								FOR j:= Iforstart TO Iforend DO
									IF NOT HMI_WorkAreaDataPicking[j].Destinazione THEN
										IF HMI_WorkAreaDataPicking[j].NumElementiDaLavorare >= 1 THEN
											ElementiDaDepositare[IdxLista] := ElementiElaborati[IdxLista] + HMI_WorkAreaDataPicking[j].NumElementiDaLavorare;
											FOR k := ElementiElaborati[IdxLista] TO ElementiDaDepositare[IdxLista]-1 DO	
												WorkAreaProductionList[NumPostazioneDeposito].PElementList[k].WA_PRELIEVO := j;
												WorkAreaProductionList[NumPostazioneDeposito].PElementList[k].WA_DEPOSITO := i;	
												ElementiElaborati[IdxLista] := ElementiElaborati[IdxLista]+1; 
											END_FOR
											CASE HMI_WorkAreaDataPicking[j].Typology OF 
												(* Se ho una cassa pianale in legno *)
												LEGNO_PIANO:
													WorkAreaState[j].Supporto.Code 					:= ActualPickingListFromHMI[IdxLista].SupportPianoLegno.Code;
													WorkAreaState[j].Supporto.DimBaseUtile		 	:= ActualPickingListFromHMI[IdxLista].SupportPianoLegno.DimBaseUtile;
													WorkAreaState[j].Supporto.AltezzaDenteRitenuta 	:= ActualPickingListFromHMI[IdxLista].SupportPianoLegno.ZDim+20;
													WorkAreaState[j].Supporto.DimVertice 			:= ActualPickingListFromHMI[IdxLista].SupportPianoLegno.DimVertice;
													WorkAreaState[j].Supporto.HMAX 					:= ActualPickingListFromHMI[IdxLista].SupportPianoLegno.HMAX;
													WorkAreaState[j].Supporto.Tipologia 			:=  e_Tipo_Pallet.CASSA_STANDARD;//ActualPickingListFromHMI[1].Support.Tipologia;
													WorkAreaState[j].Supporto.XDim 					:= ActualPickingListFromHMI[IdxLista].SupportPianoLegno.XDim;
													WorkAreaState[j].Supporto.YDim 					:= ActualPickingListFromHMI[IdxLista].SupportPianoLegno.YDim;
													WorkAreaState[j].Supporto.ZDim 					:= ActualPickingListFromHMI[IdxLista].SupportPianoLegno.ZDim;
													WorkAreaOffset[j].Y 							:= OFFSET_POSTAZIONE_LEGNO + ActualPickingListFromHMI[IdxLista].SupportPianoLegno.YDim/2;//ATTENZIONE!!! per poter lavorare in centro con i supporti pari, questa misura è la distanza tra il riscontro bundle verticale e il centro postazione PARI
												(* Se ho una cassa pianale in ferro su supporto *)
												TELAIO_PIANO:
													WorkAreaState[j].Supporto.Code 					:= ActualPickingListFromHMI[IdxLista].SupportPianoFerro.Code;
													WorkAreaState[j].Supporto.DimBaseUtile		 	:= ActualPickingListFromHMI[IdxLista].SupportPianoFerro.DimBaseUtile;
													WorkAreaState[j].Supporto.AltezzaDenteRitenuta 	:= ActualPickingListFromHMI[IdxLista].SupportPianoFerro.ZDim+20;
													WorkAreaState[j].Supporto.DimVertice 			:= ActualPickingListFromHMI[IdxLista].SupportPianoFerro.DimVertice;
													WorkAreaState[j].Supporto.HMAX 					:= ActualPickingListFromHMI[IdxLista].SupportPianoFerro.HMAX;
													WorkAreaState[j].Supporto.Tipologia 			:=  e_Tipo_Pallet.CASSA_STANDARD;//ActualPickingListFromHMI[1].Support.Tipologia;
													WorkAreaState[j].Supporto.XDim 					:= ActualPickingListFromHMI[IdxLista].SupportPianoFerro.XDim;
													WorkAreaState[j].Supporto.YDim 					:= ActualPickingListFromHMI[IdxLista].SupportPianoFerro.YDim;
													WorkAreaState[j].Supporto.ZDim 					:= ActualPickingListFromHMI[IdxLista].SupportPianoFerro.ZDim;
													WorkAreaOffset[j].Y 							:= OFFSET_POSTAZIONE_TELAIO - ActualPickingListFromHMI[IdxLista].SupportPianoFerro.YDim/2;//ATTENZIONE!!! per poter lavorare in centro con i supporti pari, questa misura è la distanza tra il riscontro bundle verticale e il centro postazione PARI
												(* Se ho un bundle *)
												BUNDLE_VERT:
													//WorkAreaState[j].P := ElementiDaDepositare;
													WorkAreaState[j].Supporto.Code 					:= ActualPickingListFromHMI[IdxLista].SupportVertBundle.Code;
													WorkAreaState[j].Supporto.DimBaseUtile		 	:= ActualPickingListFromHMI[IdxLista].SupportVertBundle.DimBaseUtile;
													WorkAreaState[j].Supporto.AltezzaDenteRitenuta 	:= ActualPickingListFromHMI[IdxLista].SupportVertBundle.ZDim+20;
													WorkAreaState[j].Supporto.DimVertice 			:= ActualPickingListFromHMI[IdxLista].SupportVertBundle.DimVertice;
													WorkAreaState[j].Supporto.HMAX 					:= ActualPickingListFromHMI[IdxLista].SupportVertBundle.HMAX;
													WorkAreaState[j].Supporto.Tipologia 			:= e_Tipo_Pallet.BUNDLE;//ActualPickingListFromHMI.SupportVertBundle.Tipologia;
													WorkAreaState[j].Supporto.XDim 					:= ActualPickingListFromHMI[IdxLista].SupportVertBundle.XDim;
													WorkAreaState[j].Supporto.YDim 					:= ActualPickingListFromHMI[IdxLista].SupportVertBundle.YDim;
													WorkAreaState[j].Supporto.ZDim 					:= ActualPickingListFromHMI[IdxLista].SupportVertBundle.ZDim;
													WorkAreaState[j].Supporto.ZDim_Ext1        		:= WorkAreaState[j].Supporto.ZDim + 20;	
													 WorkAreaOffset[j].Y 		:= 0 ;	
													//Mod 25/&/2025	  
													//WorkAreaOffset[j].Y 		:= ActualPickingListFromHMI[IdxLista].SupportVertBundle.YDim-ActualPickingListFromHMI[IdxLista].SupportVertBundle.DimBaseUtile -40;				
												(* Se ho un A_Frame *)	  
												A_FRAME_VERT:  						
													//WorkAreaState[j].P := ElementiDaDepositare;
													WorkAreaState[j].Supporto.Code 					:= ActualPickingListFromHMI[IdxLista].SupportVertCav.Code;
													WorkAreaState[j].Supporto.DimBaseUtile		 	:= ActualPickingListFromHMI[IdxLista].SupportVertCav.DimBaseUtile;
													WorkAreaState[j].Supporto.AltezzaDenteRitenuta 	:= ActualPickingListFromHMI[IdxLista].SupportVertCav.ZDim+20;
													WorkAreaState[j].Supporto.DimVertice 			:= ActualPickingListFromHMI[IdxLista].SupportVertCav.DimVertice;
													WorkAreaState[j].Supporto.HMAX 					:= ActualPickingListFromHMI[IdxLista].SupportVertcav.HMAX;
													WorkAreaState[j].Supporto.Tipologia 			:= CAVALLETTO;//ActualPickingListFromHMI.SupportVert.Tipologia;
													WorkAreaState[j].Supporto.XDim 					:= ActualPickingListFromHMI[IdxLista].SupportVertCav.XDim;
													WorkAreaState[j].Supporto.YDim 					:= ActualPickingListFromHMI[IdxLista].SupportVertCav.YDim;
													WorkAreaState[j].Supporto.ZDim 					:= ActualPickingListFromHMI[IdxLista].SupportVertCav.ZDim;
													WorkAreaState[j].Supporto.ZDim_Ext1        		:= WorkAreaState[j].Supporto.ZDim + 20;		
													WorkAreaOffset[j].Y 							:= OFFSET_POSTAZIONE_LEGNO + ActualPickingListFromHMI[IdxLista].SupportVertCav.YDim/2;//ATTENZIONE!!! per poter lavorare in centro con i supporti pari, questa misura è la distanza tra il riscontro bundle verticale e il centro postazione PARI
											   		CoordenadaPasillo0_Y := WorkArea[j].Y +  WorkAreaOffset[j].Y  - Dimensioni_Pinza.Spessore - INGOMBRO_RISCONTRO_BUNDLE - WorkAreaState[j].Supporto.YDim /2 ;
													CoordenadaPasillo180_Y := WorkArea[j].Y + WorkAreaState[j].Supporto.YDim /2 + WorkAreaOffset[j].Y  + Dimensioni_Pinza.Spessore + INGOMBRO_RISCONTRO_FRAME  ;	
											END_CASE	
											WorkAreaProductionList[j].Support := HMI_Formatura.HMI_Forming_Supporto; 
										END_IF
									END_IF     
									TFClearApprendimento(ADR(WorkAreaState[j].Apprendimento));//Azzeramento apprendimento 
								END_FOR
								EXIT; 
							(* Se ho un bundle *)
							BUNDLE_VERT:
								CASE HMI_WorkAreaDataPicking[NumPostazioneDeposito].Typology OF
									LEGNO_PIANO:
										 		WorkAreaProductionList[NumPostazioneDeposito].Support := WorkAreaState[NumPostazioneDeposito].Supporto;
												WorkAreaProductionList[NumPostazioneDeposito].Support.Tipologia	:= e_Tipo_Pallet.CASSA_STANDARD; 
									TELAIO_PIANO:
										 		WorkAreaProductionList[NumPostazioneDeposito].Support := WorkAreaState[NumPostazioneDeposito].Supporto;
												WorkAreaProductionList[NumPostazioneDeposito].Support.Tipologia	:= e_Tipo_Pallet.CASSA_STANDARD; 
									BUNDLE_VERT:
										 		WorkAreaProductionList[NumPostazioneDeposito].Support := WorkAreaState[NumPostazioneDeposito].Supporto;
												WorkAreaProductionList[NumPostazioneDeposito].Support.Tipologia	:= e_Tipo_Pallet.BUNDLE; 
									A_FRAME_VERT:
										 		WorkAreaProductionList[NumPostazioneDeposito].Support := WorkAreaState[NumPostazioneDeposito].Supporto;
												WorkAreaProductionList[NumPostazioneDeposito].Support.Tipologia	:= e_Tipo_Pallet.CAVALLETTO; 
								END_CASE
								//Se ho deposito verticale su bundle
								WorkAreaState[NumPostazioneDeposito].Supporto.Code 						:= ActualPickingListFromHMI[IdxLista].SupportVertBundle.Code;
								WorkAreaState[NumPostazioneDeposito].Supporto.DimBaseUtile		 		:= ActualPickingListFromHMI[IdxLista].SupportVertBundle.DimBaseUtile;
								WorkAreaState[NumPostazioneDeposito].Supporto.DimVertice 				:= ActualPickingListFromHMI[IdxLista].SupportVertBundle.DimVertice;
								WorkAreaState[NumPostazioneDeposito].Supporto.HMAX 						:= ActualPickingListFromHMI[IdxLista].SupportVertBundle.HMAX;
								WorkAreaState[NumPostazioneDeposito].Supporto.Tipologia 				:= e_Tipo_Pallet.BUNDLE;
								WorkAreaState[NumPostazioneDeposito].Supporto.XDim 						:= ActualPickingListFromHMI[IdxLista].SupportVertBundle.XDim;
								WorkAreaState[NumPostazioneDeposito].Supporto.YDim 						:= ActualPickingListFromHMI[IdxLista].SupportVertBundle.YDim;
								WorkAreaState[NumPostazioneDeposito].Supporto.ZDim 						:= ActualPickingListFromHMI[IdxLista].SupportVertBundle.ZDim;
								//Lo que HABIA
								//PruevaWorkAreaOffset[NumPostazioneDeposito].Y 								:= -40;	
								//Mod 25/&/2025	  
								//WorkAreaOffset[NumPostazioneDeposito].Y 								:= ActualPickingListFromHMI[IdxLista].SupportVertBundle.YDim-ActualPickingListFromHMI[IdxLista].SupportVertBundle.DimBaseUtile -20;
								FOR j:= Iforstart TO Iforend DO
									IF NOT HMI_WorkAreaDataPicking[j].Destinazione THEN
										IF HMI_WorkAreaDataPicking[j].NumElementiDaLavorare >= 1 THEN
											ElementiDaDepositare[IdxLista] := ElementiElaborati[IdxLista] + HMI_WorkAreaDataPicking[j].NumElementiDaLavorare;
											FOR k := ElementiElaborati[IdxLista] TO ElementiDaDepositare[IdxLista]-1 DO	
												WorkAreaProductionList[NumPostazioneDeposito].PElementList[k].WA_PRELIEVO := j;
												WorkAreaProductionList[NumPostazioneDeposito].PElementList[k].WA_DEPOSITO := i;	
												ElementiElaborati[IdxLista] := ElementiElaborati[IdxLista]+1; 
											END_FOR
											CASE HMI_WorkAreaDataPicking[j].Typology OF 
												(* Se ho una cassa pianale in legno *)
												LEGNO_PIANO:
													WorkAreaState[j].Supporto.Code 					:= ActualPickingListFromHMI[IdxLista].SupportPianoLegno.Code;
													WorkAreaState[j].Supporto.DimBaseUtile		 	:= ActualPickingListFromHMI[IdxLista].SupportPianoLegno.DimBaseUtile;
													WorkAreaState[j].Supporto.AltezzaDenteRitenuta 	:= ActualPickingListFromHMI[IdxLista].SupportPianoLegno.ZDim+20;
													WorkAreaState[j].Supporto.DimVertice 			:= ActualPickingListFromHMI[IdxLista].SupportPianoLegno.DimVertice;
													WorkAreaState[j].Supporto.HMAX 					:= ActualPickingListFromHMI[IdxLista].SupportPianoLegno.HMAX;
													WorkAreaState[j].Supporto.Tipologia 			:=  e_Tipo_Pallet.CASSA_STANDARD;//ActualPickingListFromHMI[1].Support.Tipologia;
													WorkAreaState[j].Supporto.XDim 					:= ActualPickingListFromHMI[IdxLista].SupportPianoLegno.XDim;
													WorkAreaState[j].Supporto.YDim 					:= ActualPickingListFromHMI[IdxLista].SupportPianoLegno.YDim;
													WorkAreaState[j].Supporto.ZDim 					:= ActualPickingListFromHMI[IdxLista].SupportPianoLegno.ZDim;
													WorkAreaOffset[j].Y 							:= OFFSET_POSTAZIONE_LEGNO + ActualPickingListFromHMI[IdxLista].SupportPianoLegno.YDim/2;//ATTENZIONE!!! per poter lavorare in centro con i supporti pari, questa misura è la distanza tra il riscontro bundle verticale e il centro postazione PARI
												(* Se ho una cassa pianale in ferro su supporto *)
												TELAIO_PIANO:
													WorkAreaState[j].Supporto.Code 					:= ActualPickingListFromHMI[IdxLista].SupportPianoFerro.Code;
													WorkAreaState[j].Supporto.DimBaseUtile		 	:= ActualPickingListFromHMI[IdxLista].SupportPianoFerro.DimBaseUtile;
													WorkAreaState[j].Supporto.AltezzaDenteRitenuta 	:= ActualPickingListFromHMI[IdxLista].SupportPianoFerro.ZDim+20;
													WorkAreaState[j].Supporto.DimVertice 			:= ActualPickingListFromHMI[IdxLista].SupportPianoFerro.DimVertice;
													WorkAreaState[j].Supporto.HMAX 					:= ActualPickingListFromHMI[IdxLista].SupportPianoFerro.HMAX;
													WorkAreaState[j].Supporto.Tipologia 			:=  e_Tipo_Pallet.CASSA_STANDARD;//ActualPickingListFromHMI[1].Support.Tipologia;
													WorkAreaState[j].Supporto.XDim 					:= ActualPickingListFromHMI[IdxLista].SupportPianoFerro.XDim;
													WorkAreaState[j].Supporto.YDim 					:= ActualPickingListFromHMI[IdxLista].SupportPianoFerro.YDim;
													WorkAreaState[j].Supporto.ZDim 					:= ActualPickingListFromHMI[IdxLista].SupportPianoFerro.ZDim;
													WorkAreaOffset[j].Y 							:= OFFSET_POSTAZIONE_TELAIO - ActualPickingListFromHMI[IdxLista].SupportPianoFerro.YDim/2;//ATTENZIONE!!! per poter lavorare in centro con i supporti pari, questa misura è la distanza tra il riscontro bundle verticale e il centro postazione PARI
												(* Se ho un bundle *)
												BUNDLE_VERT:
													//WorkAreaState[j].P := ElementiDaDepositare;
													WorkAreaState[j].Supporto.Code 					:= ActualPickingListFromHMI[IdxLista].SupportVertBundle.Code;
													WorkAreaState[j].Supporto.DimBaseUtile		 	:= ActualPickingListFromHMI[IdxLista].SupportVertBundle.DimBaseUtile;
													WorkAreaState[j].Supporto.AltezzaDenteRitenuta 	:= ActualPickingListFromHMI[IdxLista].SupportVertBundle.ZDim+20;
													WorkAreaState[j].Supporto.DimVertice 			:= ActualPickingListFromHMI[IdxLista].SupportVertBundle.DimVertice;
													WorkAreaState[j].Supporto.HMAX 					:= ActualPickingListFromHMI[IdxLista].SupportVertBundle.HMAX;
													WorkAreaState[j].Supporto.Tipologia 			:= e_Tipo_Pallet.BUNDLE;//ActualPickingListFromHMI.SupportVert.Tipologia;
													WorkAreaState[j].Supporto.XDim 					:= ActualPickingListFromHMI[IdxLista].SupportVertBundle.XDim;
													WorkAreaState[j].Supporto.YDim 					:= ActualPickingListFromHMI[IdxLista].SupportVertBundle.YDim;
													WorkAreaState[j].Supporto.ZDim 					:= ActualPickingListFromHMI[IdxLista].SupportVertBundle.ZDim;
													WorkAreaState[j].Supporto.ZDim_Ext1        		:= WorkAreaState[j].Supporto.ZDim + 20;	
													// **Lo Que Habia	
													WorkAreaOffset[j].Y 							:= 0;
													//Mod 25/&/2025	  
													//WorkAreaOffset[j].Y 		:= ActualPickingListFromHMI[IdxLista].SupportVertBundle.YDim-ActualPickingListFromHMI[IdxLista].SupportVertBundle.DimBaseUtile -40;	
			
												(* Se ho un A_Frame *)	  
												A_FRAME_VERT:  						
													//WorkAreaState[j].P := ElementiDaDepositare;
													WorkAreaState[j].Supporto.Code 					:= ActualPickingListFromHMI[IdxLista].SupportVertCav.Code;
													WorkAreaState[j].Supporto.DimBaseUtile		 	:= ActualPickingListFromHMI[IdxLista].SupportVertCav.DimBaseUtile;
													WorkAreaState[j].Supporto.AltezzaDenteRitenuta 	:= ActualPickingListFromHMI[IdxLista].SupportVertCav.ZDim+20;
													WorkAreaState[j].Supporto.DimVertice 			:= ActualPickingListFromHMI[IdxLista].SupportVertCav.DimVertice;
													WorkAreaState[j].Supporto.HMAX 					:= ActualPickingListFromHMI[IdxLista].SupportVertCav.HMAX;
													WorkAreaState[j].Supporto.Tipologia 			:= CAVALLETTO;//ActualPickingListFromHMI.SupportVert.Tipologia;
													WorkAreaState[j].Supporto.XDim 					:= ActualPickingListFromHMI[IdxLista].SupportVertCav.XDim;
													WorkAreaState[j].Supporto.YDim 					:= ActualPickingListFromHMI[IdxLista].SupportVertCav.YDim;
													WorkAreaState[j].Supporto.ZDim 					:= ActualPickingListFromHMI[IdxLista].SupportVertCav.ZDim;
													WorkAreaState[j].Supporto.ZDim_Ext1        		:= WorkAreaState[j].Supporto.ZDim + 20;		
													WorkAreaOffset[j].Y 							:= OFFSET_POSTAZIONE_LEGNO + ActualPickingListFromHMI[IdxLista].SupportVertCav.YDim/2;//ATTENZIONE!!! per poter lavorare in centro con i supporti pari, questa misura è la distanza tra il riscontro bundle verticale e il centro postazione PARI
													CoordenadaPasillo0_Y := WorkArea[j].Y +  WorkAreaOffset[j].Y  - Dimensioni_Pinza.Spessore - INGOMBRO_RISCONTRO_BUNDLE - WorkAreaState[j].Supporto.YDim /2 ;
													CoordenadaPasillo180_Y := WorkArea[j].Y + WorkAreaState[j].Supporto.YDim /2 + WorkAreaOffset[j].Y  + Dimensioni_Pinza.Spessore + INGOMBRO_RISCONTRO_FRAME  ;		  
											END_CASE
											//WorkAreaProductionList[j].Support := HMI_Formatura.HMI_Forming_Supporto;		  
											WorkAreaProductionList[j].Support := WorkAreaState[j].Supporto;
										END_IF
									END_IF
									TFClearApprendimento(ADR(WorkAreaState[j].Apprendimento));//Azzeramento apprendimento
								END_FOR
								EXIT; 
							(* Se ho un A_Frame *)	
							A_FRAME_VERT:
								WorkAreaState[NumPostazioneDeposito].Supporto.Code 						:= ActualPickingListFromHMI[IdxLista].SupportVertCav.Code;
								WorkAreaState[NumPostazioneDeposito].Supporto.DimBaseUtile		 		:= ActualPickingListFromHMI[IdxLista].SupportVertCav.DimBaseUtile;
								WorkAreaState[NumPostazioneDeposito].Supporto.DimVertice 				:= ActualPickingListFromHMI[IdxLista].SupportVertCav.DimVertice;
								WorkAreaState[NumPostazioneDeposito].Supporto.HMAX 						:= ActualPickingListFromHMI[IdxLista].SupportVertCav.HMAX;
								WorkAreaState[NumPostazioneDeposito].Supporto.Tipologia 				:= e_Tipo_Pallet.CAVALLETTO;//ActualPickingListFromHMI.SupportVertBundle.Tipologia;
								WorkAreaState[NumPostazioneDeposito].Supporto.XDim 						:= ActualPickingListFromHMI[IdxLista].SupportVertCav.XDim;
								WorkAreaState[NumPostazioneDeposito].Supporto.YDim 						:= ActualPickingListFromHMI[IdxLista].SupportVertCav.YDim;
								WorkAreaState[NumPostazioneDeposito].Supporto.ZDim 						:= ActualPickingListFromHMI[IdxLista].SupportVertCav.ZDim;
								//WorkAreaOffset[NumPostazioneDeposito].Y 								:= OFFSET_POSTAZIONE_LEGNO (*- ActualPickingListFromHMI[IdxLista].SupportPianoFerro.YDim/2*);
								WorkAreaOffset[NumPostazioneDeposito].Y 								:= OFFSET_POSTAZIONE_LEGNO + ActualPickingListFromHMI[IdxLista].SupportVertCav.YDim/2;	 
								CASE HMI_WorkAreaDataPicking[NumPostazioneDeposito].Typology OF
									LEGNO_PIANO:
										 		WorkAreaProductionList[NumPostazioneDeposito].Support := WorkAreaState[NumPostazioneDeposito].Supporto;
												WorkAreaProductionList[NumPostazioneDeposito].Support.Tipologia	:= e_Tipo_Pallet.CASSA_STANDARD; 
									TELAIO_PIANO:
										 		WorkAreaProductionList[NumPostazioneDeposito].Support := WorkAreaState[NumPostazioneDeposito].Supporto;
												WorkAreaProductionList[NumPostazioneDeposito].Support.Tipologia	:= e_Tipo_Pallet.CASSA_STANDARD; 
									BUNDLE_VERT:
										 		WorkAreaProductionList[NumPostazioneDeposito].Support := WorkAreaState[NumPostazioneDeposito].Supporto;
												WorkAreaProductionList[NumPostazioneDeposito].Support.Tipologia	:= e_Tipo_Pallet.BUNDLE; 
									A_FRAME_VERT:
										 		WorkAreaProductionList[NumPostazioneDeposito].Support := WorkAreaState[NumPostazioneDeposito].Supporto;
												WorkAreaProductionList[NumPostazioneDeposito].Support.Tipologia	:= e_Tipo_Pallet.CAVALLETTO; 
												CoordenadaPasillo0_Y := WorkArea[NumPostazioneDeposito].Y +  WorkAreaOffset[NumPostazioneDeposito].Y  - Dimensioni_Pinza.Spessore - INGOMBRO_RISCONTRO_BUNDLE - WorkAreaState[NumPostazioneDeposito].Supporto.YDim /2;
												CoordenadaPasillo180_Y := WorkArea[NumPostazioneDeposito].Y + WorkAreaState[NumPostazioneDeposito].Supporto.YDim /2 + WorkAreaOffset[NumPostazioneDeposito].Y  + Dimensioni_Pinza.Spessore + INGOMBRO_RISCONTRO_FRAME  ;		
					  
								END_CASE
								FOR j:= Iforstart TO Iforend DO
									IF NOT HMI_WorkAreaDataPicking[j].Destinazione THEN
										IF HMI_WorkAreaDataPicking[j].NumElementiDaLavorare >= 1 THEN
											ElementiDaDepositare[IdxLista] := ElementiElaborati[IdxLista] + HMI_WorkAreaDataPicking[j].NumElementiDaLavorare;
											FOR k := ElementiElaborati[IdxLista] TO ElementiDaDepositare[IdxLista]-1 DO	
												WorkAreaProductionList[NumPostazioneDeposito].PElementList[k].WA_PRELIEVO := j;
												WorkAreaProductionList[NumPostazioneDeposito].PElementList[k].WA_DEPOSITO := i;	
												ElementiElaborati[IdxLista] := ElementiElaborati[IdxLista]+1; 
											END_FOR
											CASE HMI_WorkAreaDataPicking[j].Typology OF 
												(* Se ho una cassa pianale in legno *)
												LEGNO_PIANO:
													WorkAreaState[j].Supporto.Code 					:= ActualPickingListFromHMI[IdxLista].SupportPianoLegno.Code;
													WorkAreaState[j].Supporto.DimBaseUtile		 	:= ActualPickingListFromHMI[IdxLista].SupportPianoLegno.DimBaseUtile;
													WorkAreaState[j].Supporto.AltezzaDenteRitenuta 	:= ActualPickingListFromHMI[IdxLista].SupportPianoLegno.ZDim+20;
													WorkAreaState[j].Supporto.DimVertice 			:= ActualPickingListFromHMI[IdxLista].SupportPianoLegno.DimVertice;
													WorkAreaState[j].Supporto.HMAX 					:= ActualPickingListFromHMI[IdxLista].SupportPianoLegno.HMAX;
													WorkAreaState[j].Supporto.Tipologia 			:=  e_Tipo_Pallet.CASSA_STANDARD;//ActualPickingListFromHMI[1].Support.Tipologia;
													WorkAreaState[j].Supporto.XDim 					:= ActualPickingListFromHMI[IdxLista].SupportPianoLegno.XDim;
													WorkAreaState[j].Supporto.YDim 					:= ActualPickingListFromHMI[IdxLista].SupportPianoLegno.YDim;
													WorkAreaState[j].Supporto.ZDim 					:= ActualPickingListFromHMI[IdxLista].SupportPianoLegno.ZDim;
													WorkAreaOffset[j].Y 							:= OFFSET_POSTAZIONE_LEGNO + ActualPickingListFromHMI[IdxLista].SupportPianoLegno.YDim/2;//ATTENZIONE!!! per poter lavorare in centro con i supporti pari, questa misura è la distanza tra il riscontro bundle verticale e il centro postazione PARI
												(* Se ho una cassa pianale in ferro su supporto *)
												TELAIO_PIANO:
													WorkAreaState[j].Supporto.Code 					:= ActualPickingListFromHMI[IdxLista].SupportPianoFerro.Code;
													WorkAreaState[j].Supporto.DimBaseUtile		 	:= ActualPickingListFromHMI[IdxLista].SupportPianoFerro.DimBaseUtile;
													WorkAreaState[j].Supporto.AltezzaDenteRitenuta 	:= ActualPickingListFromHMI[IdxLista].SupportPianoFerro.ZDim+20;
													WorkAreaState[j].Supporto.DimVertice 			:= ActualPickingListFromHMI[IdxLista].SupportPianoFerro.DimVertice;
													WorkAreaState[j].Supporto.HMAX 					:= ActualPickingListFromHMI[IdxLista].SupportPianoFerro.HMAX;
													WorkAreaState[j].Supporto.Tipologia 			:=  e_Tipo_Pallet.CASSA_STANDARD;//ActualPickingListFromHMI[1].Support.Tipologia;
													WorkAreaState[j].Supporto.XDim 					:= ActualPickingListFromHMI[IdxLista].SupportPianoFerro.XDim;
													WorkAreaState[j].Supporto.YDim 					:= ActualPickingListFromHMI[IdxLista].SupportPianoFerro.YDim;
													WorkAreaState[j].Supporto.ZDim 					:= ActualPickingListFromHMI[IdxLista].SupportPianoFerro.ZDim;
													WorkAreaOffset[j].Y 							:= OFFSET_POSTAZIONE_TELAIO - ActualPickingListFromHMI[IdxLista].SupportPianoFerro.YDim/2;//ATTENZIONE!!! per poter lavorare in centro con i supporti pari, questa misura è la distanza tra il riscontro bundle verticale e il centro postazione PARI
												(* Se ho un bundle *)
												BUNDLE_VERT:
													//WorkAreaState[j].P := ElementiDaDepositare;
													WorkAreaState[j].Supporto.Code 					:= ActualPickingListFromHMI[IdxLista].SupportVertBundle.Code;
													WorkAreaState[j].Supporto.DimBaseUtile		 	:= ActualPickingListFromHMI[IdxLista].SupportVertBundle.DimBaseUtile;
													WorkAreaState[j].Supporto.AltezzaDenteRitenuta 	:= ActualPickingListFromHMI[IdxLista].SupportVertBundle.ZDim+20;
													WorkAreaState[j].Supporto.DimVertice 			:= ActualPickingListFromHMI[IdxLista].SupportVertBundle.DimVertice;
													WorkAreaState[j].Supporto.HMAX 					:= ActualPickingListFromHMI[IdxLista].SupportVertBundle.HMAX;
													WorkAreaState[j].Supporto.Tipologia 			:= e_Tipo_Pallet.BUNDLE;//ActualPickingListFromHMI.SupportVert.Tipologia;
													WorkAreaState[j].Supporto.XDim 					:= ActualPickingListFromHMI[IdxLista].SupportVertBundle.XDim;
													WorkAreaState[j].Supporto.YDim 					:= ActualPickingListFromHMI[IdxLista].SupportVertBundle.YDim;
													WorkAreaState[j].Supporto.ZDim 					:= ActualPickingListFromHMI[IdxLista].SupportVertBundle.ZDim;
													WorkAreaState[j].Supporto.ZDim_Ext1        		:= WorkAreaState[j].Supporto.ZDim + 20;	
													//**Lo Que Habia
													WorkAreaOffset[j].Y 							:= 0;
													//Mod 25/&/2025	  
													//WorkAreaOffset[j].Y 		:= ActualPickingListFromHMI[IdxLista].SupportVertBundle.YDim-ActualPickingListFromHMI[IdxLista].SupportVertBundle.DimBaseUtile -40;					
												(* Se ho un A_Frame *)	  
												A_FRAME_VERT:  						
													//WorkAreaState[j].P := ElementiDaDepositare;
													WorkAreaState[j].Supporto.Code 					:= ActualPickingListFromHMI[IdxLista].SupportVertCav.Code;
													WorkAreaState[j].Supporto.DimBaseUtile		 	:= ActualPickingListFromHMI[IdxLista].SupportVertCav.DimBaseUtile;
													WorkAreaState[j].Supporto.AltezzaDenteRitenuta 	:= ActualPickingListFromHMI[IdxLista].SupportVertCav.ZDim+20;
													WorkAreaState[j].Supporto.DimVertice 			:= ActualPickingListFromHMI[IdxLista].SupportVertCav.DimVertice;
													WorkAreaState[j].Supporto.HMAX 					:= ActualPickingListFromHMI[IdxLista].SupportVertCav.HMAX;
													WorkAreaState[j].Supporto.Tipologia 			:= CAVALLETTO;//ActualPickingListFromHMI.SupportVertCav.Tipologia;
													WorkAreaState[j].Supporto.XDim 					:= ActualPickingListFromHMI[IdxLista].SupportVertCav.XDim;
													WorkAreaState[j].Supporto.YDim 					:= ActualPickingListFromHMI[IdxLista].SupportVertCav.YDim;
													WorkAreaState[j].Supporto.ZDim 					:= ActualPickingListFromHMI[IdxLista].SupportVertCav.ZDim;
													WorkAreaState[j].Supporto.ZDim_Ext1        		:= WorkAreaState[j].Supporto.ZDim + 20;		
													WorkAreaOffset[j].Y 							:= OFFSET_POSTAZIONE_LEGNO + ActualPickingListFromHMI[IdxLista].SupportVertCav.YDim/2;//ATTENZIONE!!! per poter lavorare in centro con i supporti pari, questa misura è la distanza tra il riscontro bundle verticale e il centro postazione PARI
												   CoordenadaPasillo0_Y := WorkArea[j].Y +  WorkAreaOffset[j].Y  - Dimensioni_Pinza.Spessore - INGOMBRO_RISCONTRO_BUNDLE - WorkAreaState[j].Supporto.YDim /2 ;
													CoordenadaPasillo180_Y := WorkArea[j].Y + WorkAreaState[j].Supporto.YDim /2 + WorkAreaOffset[j].Y  + Dimensioni_Pinza.Spessore + INGOMBRO_RISCONTRO_FRAME  ;	
												
											END_CASE
													  
											WorkAreaProductionList[j].Support := HMI_Formatura.HMI_Forming_Supporto;
										END_IF
									END_IF
									TFClearApprendimento(ADR(WorkAreaState[j].Apprendimento));//Azzeramento apprendimento
								END_FOR
								EXIT; 
						END_CASE // case Pricipal1
					END_IF	//-------->	 //-------> Palet destino
				END_FOR//----------For 1 HMI_WorkAreaDataPicking[i].Destinazione 
				
				Picking.Cmd_CalcolaLista[IdxLista] := TRUE;
				Temp_UDINT[8] := IdxLista;
				HMI_Forming_Attivazione[IdxLista] := TRUE;//attivo nuova formatura
			END_IF //------------------------------ActualPickingListFromHMI[IdxLista].State = e_StatoWorkOrder.DA_ESEGUIRE 
{endregion }



			Temp_UINT[9]	 := 0 ; // añadido
				 
			
			//una volta calcolata la lista per stabilire le postazioni di prelievo e quella di deposito, calcolo la formatura della postazione di deposito
			IF Picking.Cmd_CalcolaLista[IdxLista] THEN
				Temp_UINT[9]	 := IdxLista ;
				Temp_UINT[7] := j ;
				//CASE HMI_WorkAreaDataPicking[NumPostazioneDeposito].Typology OF 	 
				//CASE HMI_WorkAreaDataPicking[j].Typology OF 
				CASE HMI_WorkAreaDataPicking[NumPostazioneDeposito].Typology OF 
					TELAIO_PIANO:
						HMI_Formatura.HMI_Forming_Supporto.Code				:= RequestPickingListFromHMI[IdxLista].SupportPianoFerro.Code;
						HMI_Formatura.HMI_Forming_Supporto.XDim				:= RequestPickingListFromHMI[IdxLista].SupportPianoFerro.XDim;
						HMI_Formatura.HMI_Forming_Supporto.YDim				:= RequestPickingListFromHMI[IdxLista].SupportPianoFerro.YDim;
						HMI_Formatura.HMI_Forming_Supporto.ZDim				:= RequestPickingListFromHMI[IdxLista].SupportPianoFerro.ZDim;
						HMI_Formatura.HMI_Forming_Supporto.DimBaseUtile		:= RequestPickingListFromHMI[IdxLista].SupportPianoFerro.DimBaseUtile;
						HMI_Formatura.HMI_Forming_Supporto.DimVertice 		:= RequestPickingListFromHMI[IdxLista].SupportPianoFerro.DimVertice;
						HMI_Formatura.HMI_Forming_Supporto.HMAX 			:= RequestPickingListFromHMI[IdxLista].SupportPianoFerro.HMAX;
						HMI_Formatura.HMI_Forming_Supporto.Tipologia		:= e_Tipo_Pallet.CASSA_STANDARD;// RequestPickingListFromHMI[1].Support.Tipologia;		

					A_FRAME_VERT:
						HMI_Formatura.HMI_Forming_Supporto.Code				:= RequestPickingListFromHMI[IdxLista].SupportVertCav.Code;
						HMI_Formatura.HMI_Forming_Supporto.XDim				:= RequestPickingListFromHMI[IdxLista].SupportVertCav.XDim;
						HMI_Formatura.HMI_Forming_Supporto.YDim				:= RequestPickingListFromHMI[IdxLista].SupportVertCav.YDim;
						HMI_Formatura.HMI_Forming_Supporto.ZDim				:= RequestPickingListFromHMI[IdxLista].SupportVertCav.ZDim;
						HMI_Formatura.HMI_Forming_Supporto.TipoPianoAppoggio := 1;                      
						HMI_Formatura.HMI_Forming_Supporto.AltezzaDenteRitenuta		:= 15;              
						HMI_Formatura.HMI_Forming_Supporto.ZDim_Ext1        := HMI_Formatura.HMI_Forming_Supporto.ZDim + HMI_Formatura.HMI_Forming_Supporto.AltezzaDenteRitenuta;
						HMI_Formatura.HMI_Forming_Supporto.DimBaseUtile		:= RequestPickingListFromHMI[IdxLista].SupportVertCav.DimBaseUtile;
						HMI_Formatura.HMI_Forming_Supporto.DimVertice 		:= RequestPickingListFromHMI[IdxLista].SupportVertCav.DimVertice;
						HMI_Formatura.HMI_Forming_Supporto.HMAX 			:= RequestPickingListFromHMI[IdxLista].SupportVertCav.HMAX;
						HMI_Formatura.HMI_Forming_Supporto.Tipologia 		:= e_Tipo_Pallet.CAVALLETTO;                  
			
					BUNDLE_VERT:
						HMI_Formatura.HMI_Forming_Supporto.Code				:= RequestPickingListFromHMI[IdxLista].SupportVertBundle.Code;
						HMI_Formatura.HMI_Forming_Supporto.XDim				:= RequestPickingListFromHMI[IdxLista].SupportVertBundle.XDim;
						HMI_Formatura.HMI_Forming_Supporto.YDim				:= RequestPickingListFromHMI[IdxLista].SupportVertBundle.YDim*2;
						HMI_Formatura.HMI_Forming_Supporto.ZDim				:= RequestPickingListFromHMI[IdxLista].SupportVertBundle.ZDim;
						HMI_Formatura.HMI_Forming_Supporto.TipoPianoAppoggio := 1;                      
						HMI_Formatura.HMI_Forming_Supporto.AltezzaDenteRitenuta		:= 20;              
						HMI_Formatura.HMI_Forming_Supporto.ZDim_Ext1        := HMI_Formatura.HMI_Forming_Supporto.ZDim +	HMI_Formatura.HMI_Forming_Supporto.AltezzaDenteRitenuta;
						HMI_Formatura.HMI_Forming_Supporto.DimBaseUtile		:= RequestPickingListFromHMI[IdxLista].SupportVertBundle.DimBaseUtile;
						HMI_Formatura.HMI_Forming_Supporto.DimVertice 		:= RequestPickingListFromHMI[IdxLista].SupportVertBundle.DimVertice*2;
						HMI_Formatura.HMI_Forming_Supporto.HMAX 			:= RequestPickingListFromHMI[IdxLista].SupportVertBundle.HMAX;
						HMI_Formatura.HMI_Forming_Supporto.Tipologia 		:= e_Tipo_Pallet.BUNDLE;                  
						HMI_Formatura.HMI_Forming_Supporto.LatoDeposito 	:= 180;                     
					ELSE	
						HMI_Formatura.HMI_Forming_Supporto.Code				:= RequestPickingListFromHMI[IdxLista].SupportPianoLegno.Code;
						HMI_Formatura.HMI_Forming_Supporto.XDim				:= RequestPickingListFromHMI[IdxLista].SupportPianoLegno.XDim;
						HMI_Formatura.HMI_Forming_Supporto.YDim				:= RequestPickingListFromHMI[IdxLista].SupportPianoLegno.YDim;
						HMI_Formatura.HMI_Forming_Supporto.ZDim				:= RequestPickingListFromHMI[IdxLista].SupportPianoLegno.ZDim;
						HMI_Formatura.HMI_Forming_Supporto.DimBaseUtile		:= RequestPickingListFromHMI[IdxLista].SupportPianoLegno.DimBaseUtile;
						HMI_Formatura.HMI_Forming_Supporto.DimVertice 		:= RequestPickingListFromHMI[IdxLista].SupportPianoLegno.DimVertice;
						HMI_Formatura.HMI_Forming_Supporto.HMAX 			:= RequestPickingListFromHMI[IdxLista].SupportPianoLegno.HMAX;
						HMI_Formatura.HMI_Forming_Supporto.Tipologia		:= e_Tipo_Pallet.CASSA_STANDARD;// RequestPickingListFromHMI[1].Support.Tipologia;		
				END_CASE	
				WorkAreaProductionList[j].Support := HMI_Formatura.HMI_Forming_Supporto;		   
				//WorkAreaProductionList[NumPostazioneDeposito].Support := HMI_Formatura.HMI_Forming_Supporto;												 
				//
				HMI_Formatura.HMI_Forming_LastraDaDepositare.XDim		:= RequestPickingListFromHMI[IdxLista].SlabDimension.XDim;
				HMI_Formatura.HMI_Forming_LastraDaDepositare.YDim		:= RequestPickingListFromHMI[IdxLista].SlabDimension.YDim;
				HMI_Formatura.HMI_Forming_LastraDaDepositare.ZDim		:= RequestPickingListFromHMI[IdxLista].SlabDimension.ZDim;
																									
				HMI_Formatura.HMI_Forming_CodiciAbilitatiFormatura[IdxLista].Code[1] := 1;                 
				
				FaldaDaDepositare.TypologyCode := RequestPickingListFromHMI[IdxLista].Layer.Tipologia;
				
				FaldaDaDepositare.XDim := RequestPickingListFromHMI[IdxLista].Layer.XDim;
				FaldaDaDepositare.YDim := RequestPickingListFromHMI[IdxLista].Layer.YDim;
				FaldaDaDepositare.ZDim := RequestPickingListFromHMI[IdxLista].Layer.ZDim;
				
				//Vado ad assegnare il numero giusto di elementi a seconda se è presente o meno la falda 
				IF (RequestPickingListFromHMI[IdxLista].LayerSequence = 1 AND HMI_AbilitaDepositoFalda) AND RequestPickingListFromHMI[IdxLista].SupportPianoLegno.Tipologia <> CAVALLETTO AND RequestPickingListFromHMI[IdxLista].SupportPianoLegno.Tipologia <> BUNDLE THEN 
					HMI_Formatura.HMI_Forming_NumeroElementiDaDepositare	:= TO_UINT(2*RequestPickingListFromHMI[IdxLista].SlabNumber - 1);
				ELSE 
					HMI_Formatura.HMI_Forming_NumeroElementiDaDepositare	:= TO_UINT(RequestPickingListFromHMI[IdxLista].SlabNumber);
				END_IF
				
				//Ack 
				IF HMI_ErrAckCalcolaFormatura THEN
					HMI_Forming_ErroreCalcoli := 0;
					HMI_ErrAckCalcolaFormatura := FALSE;
					FOR i:= 1 TO MAXFORMING DO
						HMI_ConfermaAttivazioneFormatura[i] := FALSE;
						HMI_Forming_FormaturaAttivata[i] := FALSE;
					END_FOR
				END_IF
				
				//Azzeramento comandi in caso di errore
				IF HMI_Forming_ErroreCalcoli <> 0 THEN
					FOR i:=1 TO MAXFORMING DO
						HMI_Forming_Attivazione[i] 		:= FALSE;
						HMI_Forming_Disattivazione[i] 	:= FALSE;
					END_FOR
					HMI_Forming_Calcola 			:= FALSE;
				END_IF
				
				//Valorizzo altezza esterna supporto
				//IF HMI_Forming_Supporto.ZDim_Ext1 = 0 THEN
					HMI_Forming_Supporto.ZDim_Ext1 := HMI_Forming_Supporto.ZDim + HMI_Forming_Supporto.AltezzaDenteRitenuta;
				//END_IF
				//Valorizzo HMAX x tipologia pallet
				IF HMI_Forming_Supporto.Tipologia = PALLET_STANDARD THEN
					HMI_Forming_Supporto.HMAX := HMI_Forming_Supporto.ZDim;
				END_IF

				
//##########################################################################################		  
//------------------------------------------------------------------------------------------				
///////////	Attivazione	Formature  autosettata dopo caricamento dei dati dell'ordine  /////
//------------------------------------------------------------------------------------------	
					 
				//FOR i:= 1 TO MAXFORMING DO
					idxForm:= IdxLista;//forzo a 1 la formatura da attivare
					IF HMI_Forming_Attivazione[idxForm] AND idxForm <=3 AND NOT Formacion_De_listaOk[idxForm] THEN
						Forming[idxForm] := FormingEmpty;
						(*IF NOT CalcolaFormaturaTrig AND TFCalcoloFormaturaDaLista.PulisciMemoriaDone THEN *)//#Modificado
							 IF TFCalcoloFormaturaDaLista.CalcolaFormaturaDone THEN
								CalcolaFormaturaTrig := TRUE;	  
							END_IF	
						IF NOT CalcolaFormaturaTrig  AND NOT Formacion_De_listaOk[idxForm] THEN 
							HMI_Forming_FormaturaAttivata[idxForm] 	:= FALSE;
							TFCalcoloFormaturaDaLista.PulisciMemoria 	:= TRUE;
							IF TFCalcoloFormaturaDaLista.PulisciMemoriaDone THEN	
								HMI_Forming_ErroreCalcoli := 0;
								CalcolaFormaturaTrig := TRUE;
								IF (RequestPickingListFromHMI[1].LayerSequence = 0 OR NOT HMI_AbilitaDepositoFalda)
									AND HMI_Forming_NumeroElementiDaDepositare >0 
								THEN
									//Assegno l'ordine tutto a 1 perchè ho solo lastre	
									FOR i:= 1 TO MAXFORMINGSLAB DO
										//IF i <= HMI_Forming_NumeroElementiDaDepositare THEN
										IF i <= HMI_Forming_NumeroElementiDaDepositare + HMI_NumeroPezziPresentiPostazione[NumPostazioneDeposito] THEN
										//IF i <= 20THEN
											TFCalcoloFormaturaDaLista.TipoElementoDep[i] := LASTRA;//Settiamo tutte lastre!!
										ELSE
											TFCalcoloFormaturaDaLista.TipoElementoDep[i] := TERMINATORE;//Settiamo il resto come terminatore
										END_IF
									END_FOR
								ELSE
									//FOR i := 1 TO HMI_Forming_NumeroElementiDaDepositare DO//BY (Request_WorkOrder.LayerSequence+1) DO		  
									FOR i := 1 TO HMI_Forming_NumeroElementiDaDepositare DO//BY (Request_WorkOrder.LayerSequence+1) DO
										IF i MOD 2 = 1 THEN// i <= HMI_Forming_NumeroElementiDaDepositare THEN 
											TFCalcoloFormaturaDaLista.TipoElementoDep[i] := LASTRA;//Settiamo tipo lastre!!
										ELSE
											TFCalcoloFormaturaDaLista.TipoElementoDep[i] := FALDA;//Settiamo tipoi falda!
										END_IF
										TFCalcoloFormaturaDaLista.TipoElementoDep[i+1] := TERMINATORE;//Settiamo il resto come terminatore
									END_FOR
								END_IF	
								//FOR i := HMI_Forming_NumeroElementiDaDepositare+1 TO MAXFORMINGSLAB DO
								FOR i := (HMI_Forming_NumeroElementiDaDepositare + HMI_NumeroPezziPresentiPostazione[NumPostazioneDeposito] )   +1 TO MAXFORMINGSLAB DO
									TFCalcoloFormaturaDaLista.TipoElementoDep[i] := TERMINATORE;//Settiamo il resto come terminatore
								END_FOR
									
								TFCalcoloFormaturaDaLista.Materiale[e_Tipo_Elemento_Da_Lavorare.LASTRA]		:= HMI_Forming_LastraDaDepositare; 
								TFCalcoloFormaturaDaLista.Materiale[e_Tipo_Elemento_Da_Lavorare.FALDA]		:= FaldaDaDepositare;
								TFCalcoloFormaturaDaLista.Materiale[e_Tipo_Elemento_Da_Lavorare.QUADROTTA]	:= HMI_Forming_LastraDaDepositare;
								TFCalcoloFormaturaDaLista.Supporto											:= HMI_Forming_Supporto;	//Assegno la tipologia di supporto
								
								//CASE HMI_WorkAreaDataPicking[j].Typology OF //**Mod	 
								CASE HMI_WorkAreaDataPicking[NumPostazioneDeposito].Typology OF //**Mod
									BUNDLE_VERT:
										TFCalcoloFormaturaDaLista.TipoOrdinamento := 4;//Ordinamento di deposito òato 180°
									A_FRAME_VERT:
										TFCalcoloFormaturaDaLista.TipoOrdinamento := 1;//Ordinamento di deposito, prima un lato poi l'altro	
									ELSE
										TFCalcoloFormaturaDaLista.TipoOrdinamento := 2;//Ordinamento di deposito consecutivo	 
								END_CASE
									 
								TFCalcoloFormaturaDaLista.CalcolaFormatura := TRUE; 		//Lancio esecuzione dei calcoli
								MEMSET(ADR(HMI_Forming_FormaturaCalcolata),0,SIZEOF(HMI_Forming_FormaturaCalcolata));	//Pulisco la memoria di destinazione
								HMI_Forming_Attivazione[i] := FALSE;
								TFCalcoloFormaturaDaLista.PulisciMemoria := FALSE;
							END_IF
						ELSIF (TFCalcoloFormaturaDaLista.CalcolaFormaturaDone OR TFCalcoloFormaturaDaLista.Errore > 0) AND CalcolaFormaturaTrig AND NOT Formacion_De_listaOk[idxForm] THEN
							CalcolaFormaturaTrig := FALSE;
							TFCalcoloFormaturaDaLista.CalcolaFormatura := FALSE;
							Formacion_De_listaOk[idxForm] := TRUE ;
							IF TFCalcoloFormaturaDaLista.Errore = 0 THEN
								IDFormatura 								:= IDFormatura+1;
								GUIDFormatura 								:= STRING_TO_UINT(concat(UINT_TO_STRING(NUMERO_MACCHINA),UINT_TO_STRING(IDFormatura)));
								HMI_Forming_GUID 							:= GUIDFormatura;
						
								HMI_Forming_FormaturaCalcolata 				:= TFCalcoloFormaturaDaLista.FormingSlab;
								Forming[idxForm] 							:= FormingEmpty;	//Pulisco la memoria di destinazione
								Forming[idxForm] 							:= TFCalcoloFormaturaDaLista.FormingSlab;
								Forming[idxForm].Enable 					:= 1;
								Forming[idxForm].Code 						:= HMI_Forming_CodiciAbilitatiFormatura[idxForm].Code;
								Forming[idxForm].GUID						:= HMI_Forming_GUID;
								Forming[idxForm].Pallet						:= HMI_Forming_Supporto;
								HMI_Forming_IndiceFormaturaAttivata := idxForm;
								HMI_Forming_FormaturaAttivata[idxForm] 	:= TRUE;
								HMI_ConfermaAttivazioneFormatura[idxForm] := TRUE;
								//Valorizzo la struttura del WAPL per ogni elemento da elaborare
								FOR jj := 1 TO MAXELEMENTLIST DO
									IF jj < ElementiElaborati[IdxLista] THEN
										WorkAreaProductionList[NumPostazioneDeposito].PElementList[jj].PElement 		:= TFCalcoloFormaturaDaLista.FormingSlab.PElement[jj];	
										WorkAreaProductionList[NumPostazioneDeposito].PElementList[jj].Stato			:= ELEMENTO_DA_ELABORARE;
									
										IF Picking.HMI_PareggiaturaLastraAbilitata THEN
											WorkAreaProductionList[NumPostazioneDeposito].PElementList[jj].Pareggiatura := PAREGGIATURA_DA_ESEGUIRE;
										ELSE
											WorkAreaProductionList[NumPostazioneDeposito].PElementList[jj].Pareggiatura := PAREGGIATURA_DISABILITATA;
										END_IF
									ELSE
										WorkAreaProductionList[NumPostazioneDeposito].PElementList[jj].Stato			:= ELEMENTO_NOT_DEFINED;
									END_IF
								END_FOR
							ELSE
								HMI_Forming_ErroreCalcoli := TFCalcoloFormaturaDaLista.Errore;
							END_IF
							HMI_Forming_Attivazione[idxForm] := FALSE;
						END_IF
					ELSIF HMI_Forming_Attivazione[idxForm]  AND NOT Formacion_De_listaOk[idxForm] THEN
						memset(destAddr:=ADR(TFCalcoloFormaturaDaLista.Errore),fillByte:=(UINT_TO_USINT(ErrNumeroMassimoFormatureAmmesse)),n:=SIZEOF(TFCalcoloFormaturaDaLista.Errore));
					END_IF
				
					//Disattivazione formatura
					IF HMI_Forming_Disattivazione[idxForm] THEN
						HMI_Forming_Disattivazione[idxForm] := FALSE;
						Forming[idxForm] := FormingEmpty;	//Pulisco la formatura selezionata e di consegenza la disattivo
					END_IF
						
				//END_FOR
				
//####################################################################						 

						  
				(* Metto in stato di esecuzione il nuovo W.O. se tutto si è attivato *)
				IF HMI_Forming_FormaturaAttivata[IdxLista] THEN

					ActualPickingListFromHMI[IdxLista].State := e_StatoWorkOrder.DA_ESEGUIRE;
					//Azzero le liste per le postazioni dove non avviene la pallettizzazione
					FOR i:= Iforstart TO Iforend DO		 
						WorkAreaProductionList[i].Stato := e_Stato_ListaDiProduzione.LISTA_PROD_ASSENTE;
					END_FOR
					//WorkAreaProductionList[NumPostazioneDeposito].Support := Forming[idxForm].Pallet;
					WorkAreaProductionList[NumPostazioneDeposito].Stato 					:= LISTA_PROD_DA_ESEGUIRE;
					WorkAreaProductionList[NumPostazioneDeposito].NumeroListaAssociata 		:= IdxLista;
					WorkAreaState[NumPostazioneDeposito].F 									:= idxForm;
					Picking.Cmd_CalcolaLista[IdxLista] 										:= FALSE;
					HMI_Forming_FormaturaAttivata[IdxLista] 								:= FALSE;
					//CalcolaFormingRT[IdxLista] 												:= TRUE;
				END_IF
				//TFCalcoloFormaturaDaLista();
			END_IF	
		
			TFCalcoloFormaturaDaLista();
		END_IF	
		
		//verifico che la lista sia in esecuzione o terminata
		IF NOT ListaInEsecuzione[IdxLista] THEN
			FOR i:= Iforstart TO Iforend DO	
				IF WorkAreaProductionList[i].Stato = e_Stato_ListaDiProduzione.LISTA_PROD_IN_ESECUZIONE THEN
					ListaInEsecuzione[IdxLista] := TRUE;
					EXIT;	
				END_IF
			END_FOR
		ELSE
			FOR i:= Iforstart TO Iforend DO	
				IF WorkAreaProductionList[i].Stato = e_Stato_ListaDiProduzione.LISTA_PROD_ESEGUITA THEN
					ListaInEsecuzione[IdxLista] := FALSE;
					EXIT;	
				END_IF
			END_FOR
		END_IF
		
		//
		FOR i:= Iforstart TO Iforend DO	
			IF NumeroPezziPresentiPostazioneStart[i] = 0 AND WorkAreaState[i].P > 1 THEN
				NumeroPezziPresentiPostazioneStart[i] := TO_UINT(WorkAreaState[i].P);
			END_IF
		
			IF NOT HMI_WorkAreaDataPicking[i].Destinazione THEN
				IF HMI_WorkAreaDataPicking[i].NumElementiDaLavorare > 0 THEN
					//IF HMI_WorkAreaDataPicking[i].NumElementiDaLavorare >= TO_UINT(WorkAreaState[i].P)-1 THEN
					//	HMI_NumeroLastreRimanentiOrdineAttuale[i] := HMI_WorkAreaDataPicking[i].NumElementiDaLavorare - TO_UINT(WorkAreaState[i].P);
					//ELSE
					//	HMI_NumeroLastreRimanentiOrdineAttuale[i] := 0;
					//END_IF
					IF HMI_WorkAreaDataPicking[i].NumElementiDaLavorare - (TO_UINT(WorkAreaState[i].P) - NumeroPezziPresentiPostazioneStart[i]) > 0 THEN
						HMI_NumeroLastreRimanentiOrdineAttuale[i] := MIN(HMI_WorkAreaDataPicking[i].NumElementiDaLavorare,HMI_WorkAreaDataPicking[i].NumElementiDaLavorare - 
																	(NumeroPezziPresentiPostazioneStart[i] - TO_UINT(WorkAreaState[i].P)));
					ELSE
						HMI_NumeroLastreRimanentiOrdineAttuale[i] := 0;
					END_IF
				ELSE
					HMI_NumeroLastreRimanentiOrdineAttuale[i] := 0;
				END_IF
			ELSE
				IF NumeroPezziPresentiPostazioneStart[i] <= (TO_UINT(WorkAreaState[i].P)) AND NumeroPezziPresentiPostazioneStart[i]>0 THEN
					HMI_NumeroLastreRimanentiOrdineAttuale[i] := TO_UINT(WorkAreaState[i].P) - NumeroPezziPresentiPostazioneStart[i]+1;
				ELSE
					HMI_NumeroLastreRimanentiOrdineAttuale[i] := 0;
				END_IF
			END_IF
			IF (WorkAreaProductionList[i].Stato = e_Stato_ListaDiProduzione.LISTA_PROD_IN_ESECUZIONE OR WorkAreaProductionList[i].Stato = e_Stato_ListaDiProduzione.LISTA_PROD_ESEGUITA) AND WorkAreaState[i].P > 1 THEN
					//P:	(* Pack Pointer - Puntatore tabella ELEMENTO (0..n-1=, -1 dato non valido),Numero ELEMENTO successivo da depositare *)
					HMI_NumeroLastreDepOrdineAttuale[IdxLista] := TO_UINT(WorkAreaState[i].P-1);
				IF NumeroPezziPresentiPostazioneStart[i] < (TO_UINT(WorkAreaState[i].P)) AND NumeroPezziPresentiPostazioneStart[i]>0 THEN
					HMI_NumeroLastreDepOrdineAttuale[IdxLista] := TO_UINT(WorkAreaState[i].P) - NumeroPezziPresentiPostazioneStart[i];
				ELSE
					HMI_NumeroLastreDepOrdineAttuale[IdxLista] := TO_UINT(WorkAreaState[i].P) - 1;
				END_IF
			END_IF	
		END_FOR
		
		//trasferisco i valori alla variabile in lettura x HMI
		MEMCPY(destAddr:=ADR(HMI_WorkAreaProductionList),srcAddr:=ADR(WorkAreaProductionList),n:=SIZEOF(HMI_WorkAreaProductionList));
		//IF CalcolaFormingRT[IdxLista] AND NOT CalcolaFormingRT2[IdxLista] THEN //original	
			 
				  
					   
		//##################################añadido	############################################################ 
		IF 	NOT CalcolaFormingRT[IdxLista] AND NOT CalcolaFormingRT2[IdxLista] AND Temp_UINT[9] = IdxLista THEN
			
				CalcolaFormaturaTrig2 		:= FALSE ;
				CalcolaFormingRT[IdxLista] 	:= TRUE ;
	 
		END_IF
  		//#######################################################################################################
					   
							
		IF CalcolaFormingRT[IdxLista] AND NOT CalcolaFormingRT2[IdxLista] AND ActualPickingListFromHMI[IdxLista].State = 1   THEN //###############################  If  Principal calculos formaciones bendel y cabaleta
				 		//Para quitar
		Control1 := control1 +1 ;
			IF TFCalcoloFormaturaRT[IdxLista].CalcolaFormaturaDone THEN
				CalcolaFormaturaTrig2 := TRUE;	  
			END_IF
			IF NOT CalcolaFormaturaTrig2 AND NOT Formacion_bandelCalOk[idxForm]  THEN//11111111111111111
			///////////////////////////
				//CalcolaFormaturaTrig2 := TRUE;
				TFCalcoloFormaturaRT[IdxLista].PulisciMemoria 	:= TRUE;
				IF TFCalcoloFormaturaRT[IdxLista].PulisciMemoriaDone THEN		
					FOR i:= 1 TO MAXFORMINGSLAB DO
						IF i <= 40 THEN
						//IF i <= HMI_Forming_NumeroElementiDaDepositare THEN
							TFCalcoloFormaturaRT[IdxLista].TipoElementoDep[i] := LASTRA;//Settiamo tutte lastre!!
						ELSE
							TFCalcoloFormaturaRT[IdxLista].TipoElementoDep[i] := TERMINATORE;//Settiamo il resto come terminatore
						END_IF
					END_FOR
					TFCalcoloFormaturaRT[IdxLista].Materiale[e_Tipo_Elemento_Da_Lavorare.LASTRA].XDim		:= RequestPickingListFromHMI[IdxLista].SlabDimension.XDim; 
					TFCalcoloFormaturaRT[IdxLista].Materiale[e_Tipo_Elemento_Da_Lavorare.LASTRA].YDim		:= RequestPickingListFromHMI[IdxLista].SlabDimension.YDim; 
					TFCalcoloFormaturaRT[IdxLista].Materiale[e_Tipo_Elemento_Da_Lavorare.LASTRA].ZDim		:= RequestPickingListFromHMI[IdxLista].SlabDimension.ZDim; 
					TFCalcoloFormaturaRT[IdxLista].Supporto.Code											:= RequestPickingListFromHMI[IdxLista].SupportVertBundle.Code;
					TFCalcoloFormaturaRT[IdxLista].Supporto.XDim											:= RequestPickingListFromHMI[IdxLista].SupportVertBundle.XDim;
					TFCalcoloFormaturaRT[IdxLista].Supporto.YDim											:= RequestPickingListFromHMI[IdxLista].SupportVertBundle.YDim*2;
					TFCalcoloFormaturaRT[IdxLista].Supporto.ZDim				:= RequestPickingListFromHMI[IdxLista].SupportVertBundle.ZDim;
					TFCalcoloFormaturaRT[IdxLista].Supporto.TipoPianoAppoggio 	:= 1;
					TFCalcoloFormaturaRT[IdxLista].Supporto.AltezzaDenteRitenuta:= 15;
					TFCalcoloFormaturaRT[IdxLista].Supporto.ZDim_Ext1        	:= TFCalcoloFormaturaRT[IdxLista].Supporto.ZDim + TFCalcoloFormaturaRT[IdxLista].Supporto.AltezzaDenteRitenuta;
					TFCalcoloFormaturaRT[IdxLista].Supporto.DimBaseUtile		:= RequestPickingListFromHMI[IdxLista].SupportVertBundle.DimBaseUtile;
					TFCalcoloFormaturaRT[IdxLista].Supporto.DimVertice 			:= RequestPickingListFromHMI[IdxLista].SupportVertBundle.DimVertice*2;
					TFCalcoloFormaturaRT[IdxLista].Supporto.HMAX 				:= RequestPickingListFromHMI[IdxLista].SupportVertBundle.HMAX;
					TFCalcoloFormaturaRT[IdxLista].Supporto.Tipologia 			:= BUNDLE;
					TFCalcoloFormaturaRT[IdxLista].Supporto.LatoDeposito 		:= 180;
					TFCalcoloFormaturaRT[IdxLista].TipoOrdinamento				:= 4;	//Ordinamento di deposito, prima un lato poi l'altro
					TFCalcoloFormaturaRT[IdxLista].CalcolaFormatura 			:= TRUE;//Lancio esecuzione dei calcoli
					MEMSET(ADR(FormaturaBundleRT[IdxLista]),0,SIZEOF(FormaturaBundleRT[IdxLista]));	//Pulisco la memoria di destinazione
					TFCalcoloFormaturaRT[IdxLista].PulisciMemoria := FALSE;
				END_IF
			ELSIF (TFCalcoloFormaturaRT[IdxLista].CalcolaFormaturaDone OR TFCalcoloFormaturaRT[IdxLista].Errore > 0) AND CalcolaFormaturaTrig2 THEN
				CalcolaFormaturaTrig2 := FALSE;
				TFCalcoloFormaturaRT[IdxLista].CalcolaFormatura := FALSE;
				TFFormacionBandelCalculada := TFCalcoloFormaturaRT[IdxLista]; 
				FormaturaBundleRT[IdxLista] := TFCalcoloFormaturaRT[IdxLista].FormingSlab;
				IF TFCalcoloFormaturaRT[IdxLista].Errore = 0 THEN
					CalcolaFormaturaTrig2 			:= FALSE;
					CalcolaFormingRT[IdxLista] 		:= FALSE;
					CalcolaFormingRT2[IdxLista]		:= TRUE;
					Formacion_bandelCalOk[idxForm] 			:= TRUE ;
				ELSE
					CalcolaFormingRT[IdxLista] 		:= TRUE;
					CalcolaFormaturaTrig2 			:= FALSE;
				END_IF
			END_IF
		//##############################Inicio##############################################		 
		//#########################Calculo cavaleta##########################################
		ELSIF CalcolaFormingRT2[IdxLista] AND NOT CalcolaFormingRT[IdxLista] AND ActualPickingListFromHMI[IdxLista].State = 1  THEN 
			IF NOT CalcolaFormaturaTrig2 AND NOT Formacion_FrameCalOk[idxForm] THEN
			///////////////////////////
				TFCalcoloFormaturaRT[IdxLista].PulisciMemoria 	:= TRUE;	  
				
					
				//TFCalcoloFormaturaRT[IdxLista].PulisciMemoria 	:= TRUE;
				IF TFCalcoloFormaturaRT[IdxLista].PulisciMemoriaDone THEN
					CalcolaFormaturaTrig2 := TRUE;		
					FOR i:= 1 TO MAXFORMINGSLAB DO
						//IF i <= 10  THEN
						IF i <= 40 THEN
						//IF i <= HMI_Forming_NumeroElementiDaDepositare  THEN
							TFCalcoloFormaturaRT[IdxLista].TipoElementoDep[i] := LASTRA;//Settiamo tutte lastre!!
						ELSE
							TFCalcoloFormaturaRT[IdxLista].TipoElementoDep[i] := TERMINATORE;//Settiamo il resto come terminatore
						END_IF
					END_FOR
					TFCalcoloFormaturaRT[IdxLista].Materiale[e_Tipo_Elemento_Da_Lavorare.LASTRA].XDim		:= RequestPickingListFromHMI[IdxLista].SlabDimension.XDim; 
					TFCalcoloFormaturaRT[IdxLista].Materiale[e_Tipo_Elemento_Da_Lavorare.LASTRA].YDim		:= RequestPickingListFromHMI[IdxLista].SlabDimension.YDim; 
					TFCalcoloFormaturaRT[IdxLista].Materiale[e_Tipo_Elemento_Da_Lavorare.LASTRA].ZDim		:= RequestPickingListFromHMI[IdxLista].SlabDimension.ZDim; 
					TFCalcoloFormaturaRT[IdxLista].HabiCalTodasCordenadas := true ;
					TFCalcoloFormaturaRT[IdxLista].Supporto.Code											:= RequestPickingListFromHMI[IdxLista].SupportVertCav.Code;
					TFCalcoloFormaturaRT[IdxLista].Supporto.XDim											:= RequestPickingListFromHMI[IdxLista].SupportVertCav.XDim;
					TFCalcoloFormaturaRT[IdxLista].Supporto.YDim											:= RequestPickingListFromHMI[IdxLista].SupportVertCav.YDim(**2*);
					TFCalcoloFormaturaRT[IdxLista].Supporto.ZDim				:= RequestPickingListFromHMI[IdxLista].SupportVertCav.ZDim;
					TFCalcoloFormaturaRT[IdxLista].Supporto.TipoPianoAppoggio 	:= 1;
					TFCalcoloFormaturaRT[IdxLista].Supporto.AltezzaDenteRitenuta:= 13;
					TFCalcoloFormaturaRT[IdxLista].Supporto.ZDim_Ext1        	:= TFCalcoloFormaturaRT[IdxLista].Supporto.ZDim + TFCalcoloFormaturaRT[IdxLista].Supporto.AltezzaDenteRitenuta;
					TFCalcoloFormaturaRT[IdxLista].Supporto.DimBaseUtile		:= RequestPickingListFromHMI[IdxLista].SupportVertCav.DimBaseUtile;
					TFCalcoloFormaturaRT[IdxLista].Supporto.DimVertice 			:= RequestPickingListFromHMI[IdxLista].SupportVertCav.DimVertice(**2*);
					TFCalcoloFormaturaRT[IdxLista].Supporto.HMAX 				:= RequestPickingListFromHMI[IdxLista].SupportVertCav.HMAX;
					TFCalcoloFormaturaRT[IdxLista].Supporto.Tipologia 			:= CAVALLETTO;
					TFCalcoloFormaturaRT[IdxLista].Supporto.LatoDeposito 		:= 0;
					TFCalcoloFormaturaRT[IdxLista].TipoOrdinamento				:= 1;	//Ordinamento di deposito, prima un lato poi l'altro
					TFCalcoloFormaturaRT[IdxLista].CalcolaFormatura 			:= TRUE;//Lancio esecuzione dei calcoli
					MEMSET(ADR(FormaturaAFRAMERT[IdxLista]),0,SIZEOF(FormaturaAFRAMERT[IdxLista]));	//Pulisco la memoria di destinazione
					TFCalcoloFormaturaRT[IdxLista].PulisciMemoria := FALSE;
				END_IF
			ELSIF (TFCalcoloFormaturaRT[IdxLista].CalcolaFormaturaDone OR TFCalcoloFormaturaRT[IdxLista].Errore > 0) AND CalcolaFormaturaTrig2 THEN
				CalcolaFormaturaTrig2 		:= FALSE;
				TFCalcoloFormaturaRT[IdxLista].CalcolaFormatura := FALSE;
				TFFormacionCavalleteCalculada := TFCalcoloFormaturaRT[IdxLista] ;
				FormaturaAFRAMERT[IdxLista] := TFCalcoloFormaturaRT[IdxLista].FormingSlab;
				
				//CalcolaFormingRT[IdxLista] := TRUE ; // modificacion probar
				IF TFCalcoloFormaturaRT[IdxLista].Errore = 0 THEN
					CalcolaFormaturaTrig2 		:= FALSE;
					CalcolaFormingRT[IdxLista] 	:= TRUE;
					CalcolaFormingRT2[IdxLista]	:= FALSE;
					Formacion_FrameCalOk[idxForm] 		:= TRUE ;
				ELSE
					//CalcolaFormingRT[IdxLista] := TRUE; // original	  
					CalcolaFormingRT2[IdxLista] := TRUE;
				//##############################Fin ##############################################		 
				//#########################Calculo cavaleta##########################################
				END_IF
			END_IF
		END_IF //###############################  If  Principal calculos formaciones bendel y cabaleta
	
	TFCalcoloFormaturaRT[IdxLista]();
END_FOR	 
	 

	HMI_WorkAreaDataPicking_1_8 := ActualPickingListFromHMI[1].State >= 1;//Ordine postazioni 1..8 in lavoro
		 
	HMI_WorkAreaDataPicking_1_4 := (ActualPickingListFromHMI[2].State >= 1);//Ordine postazioni 1..4 in lavoro
	HMI_WorkAreaDataPicking_5_8 := (ActualPickingListFromHMI[3].State >= 1);//Ordine postazioni 5..8 in lavoro

//FOR IdxLista := 1 TO 3 DO
//	CASE IdxLista OF	 
//		1: Iforstart := 1; Iforend := MAXAREAPRESENT;
//		2: Iforstart := 1; Iforend := 4;
//		3: Iforstart := 5; Iforend := MAXAREAPRESENT;
//	END_CASE		 		   
//	FOR i:= Iforstart TO Iforend DO	
//		IF NumeroPezziPresentiPostazioneStart[i] = 0 AND WorkAreaState[i].P > 1 THEN
//			NumeroPezziPresentiPostazioneStart[i] := TO_UINT(WorkAreaState[i].P);
//		END_IF
//	
//		IF NOT HMI_WorkAreaDataPicking[i].Destinazione THEN
//			IF HMI_WorkAreaDataPicking[i].NumElementiDaLavorare > 0 THEN
//				//IF HMI_WorkAreaDataPicking[i].NumElementiDaLavorare >= TO_UINT(WorkAreaState[i].P)-1 THEN
//				//	HMI_NumeroLastreRimanentiOrdineAttuale[i] := HMI_WorkAreaDataPicking[i].NumElementiDaLavorare - TO_UINT(WorkAreaState[i].P);
//				//ELSE
//				//	HMI_NumeroLastreRimanentiOrdineAttuale[i] := 0;
//				//END_IF
//				IF HMI_WorkAreaDataPicking[i].NumElementiDaLavorare - (TO_UINT(WorkAreaState[i].P) - NumeroPezziPresentiPostazioneStart[i]) > 0 THEN
//					HMI_NumeroLastreRimanentiOrdineAttuale[i] := MIN(HMI_WorkAreaDataPicking[i].NumElementiDaLavorare,HMI_WorkAreaDataPicking[i].NumElementiDaLavorare - 
//																(NumeroPezziPresentiPostazioneStart[i] - TO_UINT(WorkAreaState[i].P)));
//				ELSE
//					HMI_NumeroLastreRimanentiOrdineAttuale[i] := 0;
//				END_IF
//			ELSE
//				HMI_NumeroLastreRimanentiOrdineAttuale[i] := 0;
//			END_IF
//		ELSE
//			IF NumeroPezziPresentiPostazioneStart[i] <= (TO_UINT(WorkAreaState[i].P)) AND NumeroPezziPresentiPostazioneStart[i]>0 THEN
//				HMI_NumeroLastreRimanentiOrdineAttuale[i] := TO_UINT(WorkAreaState[i].P) - NumeroPezziPresentiPostazioneStart[i]+1;
//			ELSE
//				HMI_NumeroLastreRimanentiOrdineAttuale[i] := 0;
//			END_IF
//		END_IF
//		IF (WorkAreaProductionList[i].Stato = e_Stato_ListaDiProduzione.LISTA_PROD_IN_ESECUZIONE OR WorkAreaProductionList[i].Stato = e_Stato_ListaDiProduzione.LISTA_PROD_ESEGUITA) AND WorkAreaState[i].P > 1 THEN
//			HMI_NumeroLastreDepOrdineAttuale[IdxLista] := TO_UINT(WorkAreaState[i].P-1);
//			IF NumeroPezziPresentiPostazioneStart[i] < (TO_UINT(WorkAreaState[i].P)) AND NumeroPezziPresentiPostazioneStart[i]>0 THEN
//				HMI_NumeroLastreDepOrdineAttuale[IdxLista] := TO_UINT(WorkAreaState[i].P) - NumeroPezziPresentiPostazioneStart[i] +1;
//			ELSE
//				HMI_NumeroLastreDepOrdineAttuale[IdxLista] := 0;
//			END_IF
//		END_IF	
//	END_FOR		  
//END_FOR			   
					
						 
							  
								   
{endregion}
END_ACTION

ACTION _11_CalcolaListaProduzioneold:
IF MachinePalletizer_TF.IN.Mode.Man AND
	(MachinePalletizer_TF.CmdExe.Code = CmdNOP OR MachinePalletizer_TF.CmdExe.Code = CmdMAN) THEN
	IF Cmd_AzzeraLista THEN
		ActualPickingListFromHMI.State := e_StatoWorkOrder.NON_ESEGUITO;
		FOR i:= 1 TO MAXAREAPRESENT DO	
			TFClearWorkAreaArray(ADR(Workarea),ADR(WorkAreaState),k:=i);
			HMI_WorkAreaDataPicking[i].Destinazione := FALSE;
			HMI_WorkAreaDataPicking[i].NumElementiDaLavorare := 0;
			WorkAreaState[i].P 			:= 1;
			WorkAreaProductionList[i] 	:= ListaEmpty;
			WorkAreaOffset[i].Y 		:= 0;
			HMI_NumeroPezziPresentiPostazione[i] := 0;
			NumeroPezziPresentiPostazioneStart[i] := 0;
		END_FOR	
		HMI_NumeroLastreDepOrdineAttuale := 0; 
		//Disattivazione formatura
		Forming[1] := FormingEmpty;	//Pulisco la formatura selezionata e di consegenza la disattivo
		ActualPickingListFromHMI.State := e_StatoWorkOrder.NON_ESEGUITO;
		//Azzero le liste per le postazioni dove non avviene la pallettizzazione
		WorkAreaProductionList[1].Stato := e_Stato_ListaDiProduzione.LISTA_PROD_ASSENTE;
		WorkAreaProductionList[2].Stato := e_Stato_ListaDiProduzione.LISTA_PROD_ASSENTE;
		WorkAreaProductionList[3].Stato := e_Stato_ListaDiProduzione.LISTA_PROD_ASSENTE;
		WorkAreaProductionList[4].Stato := e_Stato_ListaDiProduzione.LISTA_PROD_ASSENTE;
		WorkAreaProductionList[5].Stato := e_Stato_ListaDiProduzione.LISTA_PROD_ASSENTE;
		WorkAreaProductionList[6].Stato := e_Stato_ListaDiProduzione.LISTA_PROD_ASSENTE;
		WorkAreaProductionList[7].Stato := e_Stato_ListaDiProduzione.LISTA_PROD_ASSENTE;
		WorkAreaProductionList[8].Stato := e_Stato_ListaDiProduzione.LISTA_PROD_ASSENTE;
		ActualPickingListFromHMI.SlabNumber 		:= 0;
		ActualPickingListFromHMI.SlabDimension.XDim := 0;
		ActualPickingListFromHMI.SlabDimension.YDim := 0;
		ActualPickingListFromHMI.SlabDimension.ZDim := 0;
		ActualPickingListFromHMI.Support 			:= SupportDataEmpty;
		
		HMI_ErroreCalcoloLista 		:= 0;
		Picking.Cmd_CalcolaLista 	:= FALSE;
		HMI_Forming_Attivazione[1] 	:= FALSE;//attivo nuova formatura
		
		Cmd_AzzeraLista := FALSE;
		//Ack 
		//IF HMI_ErrAckCalcolaFormatura THEN
			HMI_Forming_ErroreCalcoli := 0;
			HMI_ErrAckCalcolaFormatura := FALSE;
			FOR i:= 1 TO MAXFORMING DO
				HMI_Forming_FormaturaAttivata[i] := FALSE;
			END_FOR
		//END_IF
		CalcolaFormaturaTrig := FALSE;
	END_IF
	
	IF Cmd_AttivaLista AND ActualPickingListFromHMI.State <> e_StatoWorkOrder.IN_ESECUZIONE THEN
		ElementiDaDepositare   :=0;
		HMI_ErroreCalcoloLista := 0;
		HMI_NumeroLastreDepOrdineAttuale := 0;
		FOR i:= 1 TO MAXAREAPRESENT DO	
			//HMI_WorkAreaDataPicking[i].Destinazione := FALSE;
			//HMI_WorkAreaDataPicking[i].NumElementiDaLavorare := 0;
			WorkAreaState[i].P := 1;
			WorkAreaProductionList[i] := ListaEmpty;
		END_FOR	 
		
		FOR i:= 1 TO MAXAREAPRESENT DO	
			IF NOT HMI_WorkAreaDataPicking[i].Destinazione THEN
				ElementiDaDepositare := ElementiDaDepositare+HMI_WorkAreaDataPicking[i].NumElementiDaLavorare;
				WorkAreaState[i].P := HMI_WorkAreaDataPicking[i].NumElementiDaLavorare +1;
				IF HMI_WorkAreaDataPicking[i].Vertical THEN
					WorkareaState[i].Supporto.Tipologia := BUNDLE;
				ELSE
					WorkareaState[i].Supporto.Tipologia := CASSA_STANDARD;
				END_IF
			ELSE
				NumPostazioneDeposito := i;
				HMI_WorkAreaDataPicking[NumPostazioneDeposito].NumElementiDaLavorare := RequestPickingListFromHMI.SlabNumber;
				IF HMI_WorkAreaDataPicking[i].Vertical THEN
					WorkareaState[i].Supporto.Tipologia := BUNDLE;
				ELSE
					WorkareaState[i].Supporto.Tipologia := CASSA_STANDARD;
				END_IF
			END_IF
			HMI_NumeroPezziPresentiPostazione[i] := WorkAreaState[i].P -1;
		END_FOR
	
		IF ElementiDaDepositare <= HMI_WorkAreaDataPicking[NumPostazioneDeposito].NumElementiDaLavorare THEN
			ActualPickingListFromHMI 		:= RequestPickingListFromHMI;
			ActualPickingListFromHMI.State 	:= e_StatoWorkOrder.DA_ESEGUIRE;
		ELSE
			HMI_ErroreCalcoloLista := 1;
		END_IF
		Cmd_AttivaLista 				:= FALSE;
	ELSE
		Cmd_AttivaLista 				:= FALSE;
	END_IF
	
	//attivazione lista di picking
	IF ActualPickingListFromHMI.State = e_StatoWorkOrder.DA_ESEGUIRE THEN
		ListaInEsecuzione := FALSE;
		NumeroListaInEsecuzione := 0;
	
		(* Inserimento sequenza di prelievo dalle postazioni in base al quello che l'operatore ha editato da HMI*)
		ElementiDaDepositare := 0;
		ElementiElaborati    := 1;
		NumPostazioneDeposito := 0;
		//FOR i:= 1 TO MAXAREAPRESENT DO
		//	WorkAreaState[i].P := 1;
		//END_FOR		
		
		FOR i:= 1 TO MAXAREAPRESENT DO
			IF HMI_WorkAreaDataPicking[i].Destinazione THEN
				NumPostazioneDeposito := i;
				HMI_WorkAreaDataPicking[NumPostazioneDeposito].NumElementiDaLavorare 	:= RequestPickingListFromHMI.SlabNumber;
				IF NOT HMI_WorkAreaDataPicking[NumPostazioneDeposito].Vertical THEN //Se NON ho deposito verticale
					WorkAreaState[NumPostazioneDeposito].Supporto.Code 						:= ActualPickingListFromHMI.Support.Code;
					WorkAreaState[NumPostazioneDeposito].Supporto.AltezzaDenteRitenuta 		:= ActualPickingListFromHMI.Support.DimBaseUtile;
					WorkAreaState[NumPostazioneDeposito].Supporto.DimVertice 				:= ActualPickingListFromHMI.Support.DimVertice;
					WorkAreaState[NumPostazioneDeposito].Supporto.HMAX 						:= ActualPickingListFromHMI.Support.HMAX;
					WorkAreaState[NumPostazioneDeposito].Supporto.Tipologia 				:= CASSA_STANDARD;//ActualPickingListFromHMI.Support.Tipologia;
					WorkAreaState[NumPostazioneDeposito].Supporto.XDim 						:= ActualPickingListFromHMI.Support.XDim;
					WorkAreaState[NumPostazioneDeposito].Supporto.YDim 						:= ActualPickingListFromHMI.Support.YDim;
					WorkAreaState[NumPostazioneDeposito].Supporto.ZDim 						:= ActualPickingListFromHMI.Support.ZDim;
					WorkAreaOffset[NumPostazioneDeposito].Y 								:= 1315;//ATTENZIONE!!! per poter lavorare in centro con i supporti pari, questa misura è la distanza tra il riscontro bundle verticale e il centro postazione PARI
					
					FOR j := 1 TO MAXAREAPRESENT DO
						IF NOT HMI_WorkAreaDataPicking[j].Destinazione THEN
							IF HMI_WorkAreaDataPicking[j].NumElementiDaLavorare >= 1 THEN
								ElementiDaDepositare := ElementiElaborati + HMI_WorkAreaDataPicking[j].NumElementiDaLavorare;
								FOR k := ElementiElaborati TO ElementiDaDepositare-1 DO	
									WorkAreaProductionList[NumPostazioneDeposito].PElementList[k].WA_PRELIEVO := j;
									WorkAreaProductionList[NumPostazioneDeposito].PElementList[k].WA_DEPOSITO := i;	
									ElementiElaborati := ElementiElaborati+1; 
								END_FOR
								IF NOT HMI_WorkAreaDataPicking[j].Vertical THEN
									WorkAreaState[j].Supporto.Code 					:= ActualPickingListFromHMI.Support.Code;
									WorkAreaState[j].Supporto.DimBaseUtile		 	:= ActualPickingListFromHMI.Support.DimBaseUtile;
									WorkAreaState[j].Supporto.AltezzaDenteRitenuta 	:= ActualPickingListFromHMI.Support.ZDim+20;
									WorkAreaState[j].Supporto.DimVertice 			:= ActualPickingListFromHMI.Support.DimVertice;
									WorkAreaState[j].Supporto.HMAX 					:= ActualPickingListFromHMI.Support.HMAX;
									WorkAreaState[j].Supporto.Tipologia 			:= ActualPickingListFromHMI.Support.Tipologia;
									WorkAreaState[j].Supporto.XDim 					:= ActualPickingListFromHMI.Support.XDim;
									WorkAreaState[j].Supporto.YDim 					:= ActualPickingListFromHMI.Support.YDim;
									WorkAreaState[j].Supporto.ZDim 					:= ActualPickingListFromHMI.Support.ZDim;
									WorkAreaOffset[j].Y 							:= 1315;//ATTENZIONE!!! per poter lavorare in centro con i supporti pari, questa misura è la distanza tra il riscontro bundle verticale e il centro postazione PARI
								ELSE
									//WorkAreaState[j].P := ElementiDaDepositare;
									WorkAreaState[j].Supporto.Code 					:= ActualPickingListFromHMI.SupportVert.Code;
									WorkAreaState[j].Supporto.DimBaseUtile		 	:= ActualPickingListFromHMI.SupportVert.DimBaseUtile;
									WorkAreaState[j].Supporto.AltezzaDenteRitenuta 	:= ActualPickingListFromHMI.Support.ZDim+20;
									WorkAreaState[j].Supporto.DimVertice 			:= ActualPickingListFromHMI.SupportVert.DimVertice;
									WorkAreaState[j].Supporto.HMAX 					:= ActualPickingListFromHMI.SupportVert.HMAX;
									WorkAreaState[j].Supporto.Tipologia 			:= 5;//ActualPickingListFromHMI.SupportVert.Tipologia;
									WorkAreaState[j].Supporto.XDim 					:= ActualPickingListFromHMI.SupportVert.XDim;
									WorkAreaState[j].Supporto.YDim 					:= ActualPickingListFromHMI.SupportVert.YDim;
									WorkAreaState[j].Supporto.ZDim 					:= ActualPickingListFromHMI.SupportVert.ZDim;
									WorkAreaState[j].Supporto.ZDim_Ext1        		:= WorkAreaState[j].Supporto.ZDim + 20;					
								END_IF
							END_IF
						END_IF
						TFClearApprendimento(ADR(WorkAreaState[j].Apprendimento));//Azzeramento apprendimento
					END_FOR
					EXIT; 
				ELSE //Se ho deposito verticale
					WorkAreaState[NumPostazioneDeposito].Supporto.Code 						:= ActualPickingListFromHMI.SupportVert.Code;
					WorkAreaState[NumPostazioneDeposito].Supporto.DimBaseUtile		 		:= ActualPickingListFromHMI.SupportVert.DimBaseUtile;
					WorkAreaState[NumPostazioneDeposito].Supporto.DimVertice 				:= ActualPickingListFromHMI.SupportVert.DimVertice;
					WorkAreaState[NumPostazioneDeposito].Supporto.HMAX 						:= ActualPickingListFromHMI.SupportVert.HMAX;
					WorkAreaState[NumPostazioneDeposito].Supporto.Tipologia 				:= BUNDLE;//ActualPickingListFromHMI.SupportVert.Tipologia;
					WorkAreaState[NumPostazioneDeposito].Supporto.XDim 						:= ActualPickingListFromHMI.SupportVert.XDim;
					WorkAreaState[NumPostazioneDeposito].Supporto.YDim 						:= ActualPickingListFromHMI.SupportVert.YDim;
					WorkAreaState[NumPostazioneDeposito].Supporto.ZDim 						:= ActualPickingListFromHMI.SupportVert.ZDim;
					FOR j := 1 TO MAXAREAPRESENT DO
						IF NOT HMI_WorkAreaDataPicking[j].Destinazione THEN
							IF HMI_WorkAreaDataPicking[j].NumElementiDaLavorare >= 1 THEN
								ElementiDaDepositare := ElementiElaborati + HMI_WorkAreaDataPicking[j].NumElementiDaLavorare;
								FOR k := ElementiElaborati TO ElementiDaDepositare-1 DO	
									WorkAreaProductionList[NumPostazioneDeposito].PElementList[k].WA_PRELIEVO := j;
									WorkAreaProductionList[NumPostazioneDeposito].PElementList[k].WA_DEPOSITO := i;	
									ElementiElaborati := ElementiElaborati+1; 
								END_FOR
								IF NOT HMI_WorkAreaDataPicking[j].Vertical THEN
									WorkAreaState[j].Supporto.Code 					:= ActualPickingListFromHMI.Support.Code;
									WorkAreaState[j].Supporto.DimBaseUtile		 	:= ActualPickingListFromHMI.Support.DimBaseUtile;
									WorkAreaState[j].Supporto.AltezzaDenteRitenuta 		:= ActualPickingListFromHMI.Support.ZDim+20;
									WorkAreaState[j].Supporto.DimVertice 			:= ActualPickingListFromHMI.Support.DimVertice;
									WorkAreaState[j].Supporto.HMAX 					:= ActualPickingListFromHMI.Support.HMAX;
									WorkAreaState[j].Supporto.Tipologia 			:= ActualPickingListFromHMI.Support.Tipologia;
									WorkAreaState[j].Supporto.XDim 					:= ActualPickingListFromHMI.Support.XDim;
									WorkAreaState[j].Supporto.YDim 					:= ActualPickingListFromHMI.Support.YDim;
									WorkAreaState[j].Supporto.ZDim 					:= ActualPickingListFromHMI.Support.ZDim;
									WorkAreaOffset[j].Y 							:= 1315;//ATTENZIONE!!! per poter lavorare in centro con i supporti pari, questa misura è la distanza tra il riscontro bundle verticale e il centro postazione PARI
								ELSE
									//WorkAreaState[j].P := ElementiDaDepositare;
									WorkAreaState[j].Supporto.Code 					:= ActualPickingListFromHMI.SupportVert.Code;
									WorkAreaState[j].Supporto.DimBaseUtile 			:= ActualPickingListFromHMI.SupportVert.DimBaseUtile;
									WorkAreaState[j].Supporto.AltezzaDenteRitenuta 	:= ActualPickingListFromHMI.Support.ZDim+20;
									WorkAreaState[j].Supporto.DimVertice 			:= ActualPickingListFromHMI.SupportVert.DimVertice;
									WorkAreaState[j].Supporto.HMAX 					:= ActualPickingListFromHMI.SupportVert.HMAX;
									WorkAreaState[j].Supporto.Tipologia 			:= 5;//ActualPickingListFromHMI.SupportVert.Tipologia;
									WorkAreaState[j].Supporto.XDim 					:= ActualPickingListFromHMI.SupportVert.XDim;
									WorkAreaState[j].Supporto.YDim 					:= ActualPickingListFromHMI.SupportVert.YDim;
									WorkAreaState[j].Supporto.ZDim 					:= ActualPickingListFromHMI.SupportVert.ZDim;
									WorkAreaState[j].Supporto.ZDim_Ext1        		:= WorkAreaState[j].Supporto.ZDim + 20;
								END_IF
							END_IF
						END_IF
						TFClearApprendimento(ADR(WorkAreaState[j].Apprendimento));//Azzeramento apprendimento
					END_FOR
					EXIT; 
				END_IF
			END_IF
		END_FOR
		
		Picking.Cmd_CalcolaLista := TRUE;
		HMI_Forming_Attivazione[1] := TRUE;//attivo nuova formatura
	END_IF
	
	//una volta calcolata la lista per stabilire le postazioni di prelievo e quella di deposito, calcolo la formatura della postazione di deposito
	IF Picking.Cmd_CalcolaLista THEN
		IF NOT HMI_WorkAreaDataPicking[NumPostazioneDeposito].Vertical THEN
			HMI_Formatura.HMI_Forming_Supporto.Code				:= RequestPickingListFromHMI.Support.Code;
			HMI_Formatura.HMI_Forming_Supporto.XDim				:= RequestPickingListFromHMI.Support.XDim;
			HMI_Formatura.HMI_Forming_Supporto.YDim				:= RequestPickingListFromHMI.Support.YDim;
			HMI_Formatura.HMI_Forming_Supporto.ZDim				:= RequestPickingListFromHMI.Support.ZDim;
			HMI_Formatura.HMI_Forming_Supporto.DimBaseUtile		:= RequestPickingListFromHMI.Support.DimBaseUtile;
			HMI_Formatura.HMI_Forming_Supporto.DimVertice 		:= RequestPickingListFromHMI.Support.DimVertice;
			HMI_Formatura.HMI_Forming_Supporto.HMAX 			:= RequestPickingListFromHMI.Support.HMAX;
			HMI_Formatura.HMI_Forming_Supporto.Tipologia		:= RequestPickingListFromHMI.Support.Tipologia;
		ELSE
			HMI_Formatura.HMI_Forming_Supporto.Code				:= RequestPickingListFromHMI.SupportVert.Code;
			HMI_Formatura.HMI_Forming_Supporto.XDim				:= RequestPickingListFromHMI.Supportvert.XDim;
			HMI_Formatura.HMI_Forming_Supporto.YDim				:= RequestPickingListFromHMI.Supportvert.YDim*2;
			HMI_Formatura.HMI_Forming_Supporto.ZDim				:= RequestPickingListFromHMI.Supportvert.ZDim;
			HMI_Formatura.HMI_Forming_Supporto.TipoPianoAppoggio := 1;
			HMI_Formatura.HMI_Forming_Supporto.AltezzaDenteRitenuta		:= 20;
			HMI_Formatura.HMI_Forming_Supporto.ZDim_Ext1        := HMI_Formatura.HMI_Forming_Supporto.ZDim +	HMI_Formatura.HMI_Forming_Supporto.AltezzaDenteRitenuta;
			HMI_Formatura.HMI_Forming_Supporto.DimBaseUtile		:= RequestPickingListFromHMI.Supportvert.DimBaseUtile;
			HMI_Formatura.HMI_Forming_Supporto.DimVertice 		:= RequestPickingListFromHMI.Supportvert.DimVertice*2;
			HMI_Formatura.HMI_Forming_Supporto.HMAX 			:= RequestPickingListFromHMI.Supportvert.HMAX;
			HMI_Formatura.HMI_Forming_Supporto.Tipologia 		:= BUNDLE;
			HMI_Formatura.HMI_Forming_Supporto.LatoDeposito 	:= 180;
		END_IF
		//
		HMI_Formatura.HMI_Forming_LastraDaDepositare.XDim		:= RequestPickingListFromHMI.SlabDimension.XDim;
		HMI_Formatura.HMI_Forming_LastraDaDepositare.YDim		:= RequestPickingListFromHMI.SlabDimension.YDim;
		HMI_Formatura.HMI_Forming_LastraDaDepositare.ZDim		:= RequestPickingListFromHMI.SlabDimension.ZDim;
		
		HMI_Formatura.HMI_Forming_CodiciAbilitatiFormatura[1].Code[1] := 1;
		
		FaldaDaDepositare.TypologyCode := RequestPickingListFromHMI.Layer.Tipologia;
		
		FaldaDaDepositare.XDim := RequestPickingListFromHMI.Layer.XDim;
		FaldaDaDepositare.YDim := RequestPickingListFromHMI.Layer.YDim;
		FaldaDaDepositare.ZDim := RequestPickingListFromHMI.Layer.ZDim;
		
		//Vado ad assegnare il numero giusto di elementi a seconda se è presente o meno la falda 
		IF (RequestPickingListFromHMI.LayerSequence = 1 AND HMI_AbilitaDepositoFalda) AND RequestPickingListFromHMI.Support.Tipologia <> CAVALLETTO AND RequestPickingListFromHMI.Support.Tipologia <> BUNDLE THEN 
			HMI_Formatura.HMI_Forming_NumeroElementiDaDepositare	:= TO_UINT(2*RequestPickingListFromHMI.SlabNumber - 1);
		ELSE 
			HMI_Formatura.HMI_Forming_NumeroElementiDaDepositare	:= TO_UINT(RequestPickingListFromHMI.SlabNumber);
		END_IF
		
		//Ack 
		IF HMI_ErrAckCalcolaFormatura THEN
			HMI_Forming_ErroreCalcoli := 0;
			HMI_ErrAckCalcolaFormatura := FALSE;
			FOR i:= 1 TO MAXFORMING DO
				HMI_Forming_FormaturaAttivata[i] := FALSE;
			END_FOR
		END_IF
		
		//Azzeramento comandi in caso di errore
		IF HMI_Forming_ErroreCalcoli <> 0 THEN
			FOR i:=1 TO MAXFORMING DO
				HMI_Forming_Attivazione[i] 		:= FALSE;
				HMI_Forming_Disattivazione[i] 	:= FALSE;
			END_FOR
			HMI_Forming_Calcola 			:= FALSE;
		END_IF
		
		//Valorizzo altezza esterna supporto
		//IF HMI_Forming_Supporto.ZDim_Ext1 = 0 THEN
			HMI_Forming_Supporto.ZDim_Ext1 := HMI_Forming_Supporto.ZDim + HMI_Forming_Supporto.AltezzaDenteRitenuta;
		//END_IF
		//Valorizzo HMAX x tipologia pallet
		IF HMI_Forming_Supporto.Tipologia = PALLET_STANDARD THEN
			HMI_Forming_Supporto.HMAX := HMI_Forming_Supporto.ZDim;
		END_IF
		
		//Attivazione
		//FOR i:= 1 TO MAXFORMING DO
			idxForm:=1;//forzo a 1 la formatura da attivare
			IF HMI_Forming_Attivazione[idxForm] AND idxForm <=2 THEN
				Forming[idxForm] := FormingEmpty;
				IF NOT CalcolaFormaturaTrig  THEN
					HMI_Forming_FormaturaAttivata[idxForm] 	:= FALSE;
					TFCalcoloFormaturaDaLista.PulisciMemoria 	:= TRUE;
					IF TFCalcoloFormaturaDaLista.PulisciMemoriaDone THEN	
						HMI_Forming_ErroreCalcoli := 0;
						
						IF RequestPickingListFromHMI.LayerSequence = 0 OR NOT HMI_AbilitaDepositoFalda THEN
							//Assegno l'ordine tutto a 1 perchè ho solo lastre	
							FOR i:= 1 TO MAXFORMINGSLAB DO
								IF i <= HMI_Forming_NumeroElementiDaDepositare THEN
									TFCalcoloFormaturaDaLista.TipoElementoDep[i] := LASTRA;//Settiamo tutte lastre!!
								ELSE
									TFCalcoloFormaturaDaLista.TipoElementoDep[i] := TERMINATORE;//Settiamo il resto come terminatore
								END_IF
							END_FOR
						ELSE
							FOR i := 1 TO HMI_Forming_NumeroElementiDaDepositare DO//BY (Request_WorkOrder.LayerSequence+1) DO
								IF i MOD 2 = 1 THEN// i <= HMI_Forming_NumeroElementiDaDepositare THEN 
									TFCalcoloFormaturaDaLista.TipoElementoDep[i] := LASTRA;//Settiamo tipo lastre!!
								ELSE
									TFCalcoloFormaturaDaLista.TipoElementoDep[i] := FALDA;//Settiamo tipoi falda!
								END_IF
								TFCalcoloFormaturaDaLista.TipoElementoDep[i+1] := TERMINATORE;//Settiamo il resto come terminatore
							END_FOR
						END_IF	
						FOR i := HMI_Forming_NumeroElementiDaDepositare+1 TO MAXFORMINGSLAB DO
							TFCalcoloFormaturaDaLista.TipoElementoDep[i] := TERMINATORE;//Settiamo il resto come terminatore
						END_FOR
							
						TFCalcoloFormaturaDaLista.Materiale[e_Tipo_Elemento_Da_Lavorare.LASTRA]		:= HMI_Forming_LastraDaDepositare; 
						TFCalcoloFormaturaDaLista.Materiale[e_Tipo_Elemento_Da_Lavorare.FALDA]		:= FaldaDaDepositare;
						TFCalcoloFormaturaDaLista.Materiale[e_Tipo_Elemento_Da_Lavorare.QUADROTTA]	:= HMI_Forming_LastraDaDepositare;
						TFCalcoloFormaturaDaLista.Supporto											:= HMI_Forming_Supporto;	//Assegno la tipologia di supporto
						IF HMI_WorkAreaDataPicking[NumPostazioneDeposito].Vertical THEN//Se sono in deposito verticale -> sono sul bundle...
							TFCalcoloFormaturaDaLista.TipoOrdinamento									:= 4;//Ordinamento di deposito, prima un lato poi l'altro
						ELSE
							TFCalcoloFormaturaDaLista.TipoOrdinamento									:= 2;//Ordinamento di deposito, prima un lato poi l'altro
						END_IF
						TFCalcoloFormaturaDaLista.CalcolaFormatura := TRUE; 		//Lancio esecuzione dei calcoli
						MEMSET(ADR(HMI_Forming_FormaturaCalcolata),0,SIZEOF(HMI_Forming_FormaturaCalcolata));	//Pulisco la memoria di destinazione
						CalcolaFormaturaTrig := TRUE;
						HMI_Forming_Attivazione[i] := FALSE;
						TFCalcoloFormaturaDaLista.PulisciMemoria := FALSE;
					END_IF
				ELSIF (TFCalcoloFormaturaDaLista.CalcolaFormaturaDone OR TFCalcoloFormaturaDaLista.Errore > 0) AND CalcolaFormaturaTrig THEN
					TFCalcoloFormaturaDaLista.CalcolaFormatura := FALSE;
					IF TFCalcoloFormaturaDaLista.Errore = 0 THEN
						IDFormatura 			:= IDFormatura+1;
						GUIDFormatura 			:= STRING_TO_UINT(concat(UINT_TO_STRING(NUMERO_MACCHINA),UINT_TO_STRING(IDFormatura)));
						HMI_Forming_GUID 		:= GUIDFormatura;
				
						HMI_Forming_FormaturaCalcolata 		:= TFCalcoloFormaturaDaLista.FormingSlab;
						Forming[idxForm] 							:= FormingEmpty;	//Pulisco la memoria di destinazione
						Forming[idxForm] 							:= TFCalcoloFormaturaDaLista.FormingSlab;
						Forming[idxForm].Enable 					:= 1;
						Forming[idxForm].Code 					:= HMI_Forming_CodiciAbilitatiFormatura[idxForm].Code;
						Forming[idxForm].GUID						:= HMI_Forming_GUID;
						Forming[idxForm].Pallet					:= HMI_Forming_Supporto;
						HMI_Forming_IndiceFormaturaAttivata := idxForm;
						HMI_Forming_FormaturaAttivata[idxForm] 	:= TRUE;
						//Valorizzo la struttura del WAPL per ogni elemento da elaborare
						FOR j := 1 TO MAXELEMENTLIST DO
							IF j < ElementiElaborati THEN
								WorkAreaProductionList[NumPostazioneDeposito].PElementList[j].PElement 		:= TFCalcoloFormaturaDaLista.FormingSlab.PElement[j];	
								WorkAreaProductionList[NumPostazioneDeposito].PElementList[j].Stato			:= ELEMENTO_DA_ELABORARE;
							
								IF Picking.HMI_PareggiaturaLastraAbilitata THEN
									WorkAreaProductionList[NumPostazioneDeposito].PElementList[j].Pareggiatura := PAREGGIATURA_DA_ESEGUIRE;
								ELSE
									WorkAreaProductionList[NumPostazioneDeposito].PElementList[j].Pareggiatura := PAREGGIATURA_DISABILITATA;
								END_IF
							ELSE
								WorkAreaProductionList[NumPostazioneDeposito].PElementList[j].Stato			:= ELEMENTO_NOT_DEFINED;
							END_IF
						END_FOR
					ELSE
						HMI_Forming_ErroreCalcoli := TFCalcoloFormaturaDaLista.Errore;
					END_IF
					CalcolaFormaturaTrig := FALSE;
					HMI_Forming_Attivazione[idxForm] := FALSE;
				END_IF
			ELSIF HMI_Forming_Attivazione[idxForm] THEN
				memset(destAddr:=ADR(TFCalcoloFormaturaDaLista.Errore),fillByte:=(UINT_TO_USINT(ErrNumeroMassimoFormatureAmmesse)),n:=SIZEOF(TFCalcoloFormaturaDaLista.Errore));
			END_IF
		
			//Disattivazione formatura
			IF HMI_Forming_Disattivazione[idxForm] THEN
				HMI_Forming_Disattivazione[idxForm] := FALSE;
				Forming[idxForm] := FormingEmpty;	//Pulisco la formatura selezionata e di consegenza la disattivo
			END_IF
				
		//END_FOR
		
		(* Metto in stato di esecuzione il nuovo W.O. se tutto si è attivato *)
		IF HMI_Forming_FormaturaAttivata[1] THEN
			ActualPickingListFromHMI.State := e_StatoWorkOrder.IN_ESECUZIONE;
			//Azzero le liste per le postazioni dove non avviene la pallettizzazione
			WorkAreaProductionList[1].Stato := e_Stato_ListaDiProduzione.LISTA_PROD_ASSENTE;
			WorkAreaProductionList[2].Stato := e_Stato_ListaDiProduzione.LISTA_PROD_ASSENTE;
			WorkAreaProductionList[3].Stato := e_Stato_ListaDiProduzione.LISTA_PROD_ASSENTE;
			WorkAreaProductionList[4].Stato := e_Stato_ListaDiProduzione.LISTA_PROD_ASSENTE;
			WorkAreaProductionList[5].Stato := e_Stato_ListaDiProduzione.LISTA_PROD_ASSENTE;
			WorkAreaProductionList[6].Stato := e_Stato_ListaDiProduzione.LISTA_PROD_ASSENTE;
			WorkAreaProductionList[7].Stato := e_Stato_ListaDiProduzione.LISTA_PROD_ASSENTE;
			WorkAreaProductionList[8].Stato := e_Stato_ListaDiProduzione.LISTA_PROD_ASSENTE;
			WorkAreaProductionList[NumPostazioneDeposito].Support := Forming[idxForm].Pallet;
			WorkAreaProductionList[NumPostazioneDeposito].Stato := LISTA_PROD_DA_ESEGUIRE;
			Picking.Cmd_CalcolaLista := FALSE;
			HMI_Forming_FormaturaAttivata[1] := FALSE;
			CalcolaFormingRT := TRUE;
		END_IF
	END_IF	
	TFCalcoloFormaturaDaLista();
END_IF	

//verifico che la lista sia in esecuzione o terminata
IF NOT ListaInEsecuzione THEN
	FOR i := 1 TO MAXAREAPRESENT DO	
		IF WorkAreaProductionList[i].Stato = e_Stato_ListaDiProduzione.LISTA_PROD_IN_ESECUZIONE THEN
			ListaInEsecuzione := TRUE;
			EXIT;	
		END_IF
	END_FOR
ELSE
	FOR i := 1 TO MAXAREAPRESENT DO	
		IF WorkAreaProductionList[i].Stato = e_Stato_ListaDiProduzione.LISTA_PROD_ESEGUITA THEN
			ListaInEsecuzione := FALSE;
			EXIT;	
		END_IF
	END_FOR
END_IF

//



FOR i := 1 TO MAXAREAPRESENT DO	
		
	IF NumeroPezziPresentiPostazioneStart[i] = 0 AND WorkAreaState[i].P > 1 THEN
		NumeroPezziPresentiPostazioneStart[i] := TO_UINT(WorkAreaState[i].P);
	END_IF

	IF NOT HMI_WorkAreaDataPicking[i].Destinazione THEN
		IF HMI_WorkAreaDataPicking[i].NumElementiDaLavorare > 0 THEN
			//IF HMI_WorkAreaDataPicking[i].NumElementiDaLavorare >= TO_UINT(WorkAreaState[i].P)-1 THEN
			//	HMI_NumeroLastreRimanentiOrdineAttuale[i] := HMI_WorkAreaDataPicking[i].NumElementiDaLavorare - TO_UINT(WorkAreaState[i].P);
			//ELSE
			//	HMI_NumeroLastreRimanentiOrdineAttuale[i] := 0;
			//END_IF
			IF HMI_WorkAreaDataPicking[i].NumElementiDaLavorare - (TO_UINT(WorkAreaState[i].P) - NumeroPezziPresentiPostazioneStart[i]) > 0 THEN
				HMI_NumeroLastreRimanentiOrdineAttuale[i] := MIN(HMI_WorkAreaDataPicking[i].NumElementiDaLavorare,HMI_WorkAreaDataPicking[i].NumElementiDaLavorare - 
															(NumeroPezziPresentiPostazioneStart[i] - TO_UINT(WorkAreaState[i].P)));
			ELSE
				HMI_NumeroLastreRimanentiOrdineAttuale[i] := 0;
			END_IF
		ELSE
			HMI_NumeroLastreRimanentiOrdineAttuale[i] := 0;
		END_IF
	ELSE
		IF NumeroPezziPresentiPostazioneStart[i] < (TO_UINT(WorkAreaState[i].P)) AND NumeroPezziPresentiPostazioneStart[i]>0 THEN
			HMI_NumeroLastreRimanentiOrdineAttuale[i] := TO_UINT(WorkAreaState[i].P) - NumeroPezziPresentiPostazioneStart[i]+1;
		ELSE
			HMI_NumeroLastreRimanentiOrdineAttuale[i] := 0;
		END_IF
	END_IF
	IF (WorkAreaProductionList[i].Stato = e_Stato_ListaDiProduzione.LISTA_PROD_IN_ESECUZIONE OR WorkAreaProductionList[i].Stato = e_Stato_ListaDiProduzione.LISTA_PROD_ESEGUITA) AND WorkAreaState[i].P > 1 THEN
		HMI_NumeroLastreDepOrdineAttuale := TO_UINT(WorkAreaState[i].P-1);
		IF NumeroPezziPresentiPostazioneStart[i] < (TO_UINT(WorkAreaState[i].P)) AND NumeroPezziPresentiPostazioneStart[i]>0 THEN
			HMI_NumeroLastreDepOrdineAttuale := TO_UINT(WorkAreaState[i].P) - NumeroPezziPresentiPostazioneStart[i];
		ELSE
			HMI_NumeroLastreDepOrdineAttuale := 0;
		END_IF
	END_IF	
END_FOR

//trasferisco i valori alla variabile in lettura x HMI
MEMCPY(destAddr:=ADR(HMI_WorkAreaProductionList),srcAddr:=ADR(WorkAreaProductionList),n:=SIZEOF(HMI_WorkAreaProductionList));
	
IF CalcolaFormingRT THEN
	IF NOT CalcolaFormaturaTrig2 THEN
	///////////////////////////
		TFCalcoloFormaturaRT.PulisciMemoria 	:= TRUE;
		IF TFCalcoloFormaturaRT.PulisciMemoriaDone THEN		
			FOR i:= 1 TO MAXFORMINGSLAB DO
				IF i <= 50 THEN
					TFCalcoloFormaturaRT.TipoElementoDep[i] := LASTRA;//Settiamo tutte lastre!!
				ELSE
					TFCalcoloFormaturaRT.TipoElementoDep[i] := TERMINATORE;//Settiamo il resto come terminatore
				END_IF
			END_FOR
			TFCalcoloFormaturaRT.Materiale[e_Tipo_Elemento_Da_Lavorare.LASTRA].XDim		:= RequestPickingListFromHMI.SlabDimension.XDim; 
			TFCalcoloFormaturaRT.Materiale[e_Tipo_Elemento_Da_Lavorare.LASTRA].YDim		:= RequestPickingListFromHMI.SlabDimension.YDim; 
			TFCalcoloFormaturaRT.Materiale[e_Tipo_Elemento_Da_Lavorare.LASTRA].ZDim		:= RequestPickingListFromHMI.SlabDimension.ZDim; 
			TFCalcoloFormaturaRT.Supporto.Code					:= RequestPickingListFromHMI.SupportVert.Code;
			TFCalcoloFormaturaRT.Supporto.XDim					:= RequestPickingListFromHMI.Supportvert.XDim;
			TFCalcoloFormaturaRT.Supporto.YDim					:= RequestPickingListFromHMI.Supportvert.YDim*2;
			TFCalcoloFormaturaRT.Supporto.ZDim					:= RequestPickingListFromHMI.Supportvert.ZDim;
			TFCalcoloFormaturaRT.Supporto.TipoPianoAppoggio 	:= 1;
			TFCalcoloFormaturaRT.Supporto.AltezzaDenteRitenuta	:= 20;
			TFCalcoloFormaturaRT.Supporto.ZDim_Ext1        	:= TFCalcoloFormaturaRT.Supporto.ZDim + TFCalcoloFormaturaRT.Supporto.AltezzaDenteRitenuta;
			TFCalcoloFormaturaRT.Supporto.DimBaseUtile		:= RequestPickingListFromHMI.Supportvert.DimBaseUtile;
			TFCalcoloFormaturaRT.Supporto.DimVertice 		:= RequestPickingListFromHMI.Supportvert.DimVertice*2;
			TFCalcoloFormaturaRT.Supporto.HMAX 				:= RequestPickingListFromHMI.Supportvert.HMAX;
			TFCalcoloFormaturaRT.Supporto.Tipologia 		:= BUNDLE;
			TFCalcoloFormaturaRT.Supporto.LatoDeposito 		:= 180;
			TFCalcoloFormaturaRT.TipoOrdinamento			:= 4;//Ordinamento di deposito, prima un lato poi l'altro
			TFCalcoloFormaturaRT.CalcolaFormatura := TRUE; 		//Lancio esecuzione dei calcoli
			MEMSET(ADR(FormaturaRT),0,SIZEOF(FormaturaRT));	//Pulisco la memoria di destinazione
			CalcolaFormaturaTrig2 := TRUE;
			TFCalcoloFormaturaRT.PulisciMemoria := FALSE;
		END_IF
	ELSIF (TFCalcoloFormaturaRT.CalcolaFormaturaDone OR TFCalcoloFormaturaRT.Errore > 0) AND CalcolaFormaturaTrig2 THEN
		TFCalcoloFormaturaRT.CalcolaFormatura := FALSE;
		FormaturaRT := TFCalcoloFormaturaRT.FormingSlab;
		CalcolaFormaturaTrig2 := FALSE;
		IF TFCalcoloFormaturaRT.Errore = 0 THEN
			CalcolaFormaturaTrig2 := FALSE;
			CalcolaFormingRT := FALSE;
		ELSE
			CalcolaFormingRT := TRUE;;
		END_IF
	END_IF
END_IF
TFCalcoloFormaturaRT();
END_ACTION

ACTION TEST_Variabili:

	Temp_Bool[8] := MachinePalletizer_TF.OUT.ClockSegnalazioni;
	Temp_Bool[9] := MachinePalletizer_TF.OUT.ClockSegnalazioniAlternato;

	Temp_Bool[0] := HMI_Status_BarrieraPall_OK;

  
 Temp_uint[0] := ElementiDaDepositare[1];	
 Temp_uint[0] := ElementiDaDepositare[2];		
 Temp_uint[0] := ElementiDaDepositare[3];
		 
 Temp_uint[0] := HMI_WorkAreaDataPicking[1].NumElementiDaLavorare;	
 Temp_uint[0] := HMI_WorkAreaDataPicking[1].NumElementiDaLavorare;		

	
 Temp_Real[1]:= 	MachinePalletizer_TF.WorkSpace[1].X;
 Temp_Real[1]:= 	MachinePalletizer_TF.WorkSpace[1].Y;
 Temp_Real[1]:= 	MachinePalletizer_TF.WorkSpace[1].Z;
   
 
 Temp_Real[1]:= Traiettoria.StartPoint.X;
 Temp_Real[1]:= Traiettoria.StartPoint.Y;
 Temp_Real[1]:= Traiettoria.StartPoint.Z;
 Temp_Real[1]:= Traiettoria.StartPoint.J;


//; SimulazioneSenzaPalletFalde;
//PINZA
Temp_Real[1]:= Pinza.Ovem1.Status.ValoreDepressioneIstantanea;
Temp_Real[1]:= HMI_DepressioneOVEM_DX1;
Temp_Real[1]:= Pinza.Ovem12.Status.ValoreDepressioneIstantanea;
Temp_Real[1]:= HMI_DepressioneOVEM_DX2;
//;
Temp_Real[1]:= Pinza.Ovem22.Status.ValoreDepressioneIstantanea;
Temp_Real[1]:= HMI_DepressioneOVEM_SX1;
Temp_Real[1]:= Pinza.Ovem22.Status.ValoreDepressioneIstantanea;
Temp_Real[1]:= HMI_DepressioneOVEM_SX2;
	
//Presenza
//FormaturaAFRAMERT;
Temp_bool[0] := I_PresenzaSupporto[1];
Temp_bool[0] := I_PresenzaBundle[1];
Temp_bool[0] := I_PresenzaCentrale[1];
Temp_bool[0] := I_PHPresenzaPallet[1];
Temp_bool[0] := I_PHPresenzaPalletVirtuale[1];

Temp_bool[0] := I_PresenzaSupporto[2];
Temp_bool[0] := I_PresenzaBundle[2];
Temp_bool[0] := I_PresenzaCentrale[2];
Temp_bool[0] := I_PHPresenzaPallet[2];
Temp_bool[0] := I_PHPresenzaPalletVirtuale[2];

Temp_bool[0] := I_PresenzaSupporto[3];
Temp_bool[0] := I_PresenzaBundle[3];
Temp_bool[0] := I_PresenzaCentrale[3];
Temp_bool[0] := I_PHPresenzaPallet[3];
Temp_bool[0] := I_PHPresenzaPalletVirtuale[3];

//*** Calcola Lista produzione  ***	

 Temp_bool[0] := HMI_WorkAreaDataPicking[1].Destinazione; // (0=Prelievo, 1= deposito).	
 Temp_bool[0] := HMI_WorkAreaDataPicking[2].Destinazione;
 Temp_bool[0] := HMI_WorkAreaDataPicking[3].Destinazione;
 Temp_bool[0] := HMI_WorkAreaDataPicking[4].Destinazione;
 
//valori dei supporti della lista 2
Temp_Real[1]:= RequestPickingListFromHMI[2].SupportPianoLegno.XDim;
Temp_Real[1]:= RequestPickingListFromHMI[2].SupportPianoLegno.YDim;	
Temp_real[1]:= RequestPickingListFromHMI[2].SupportPianoLegno.ZDim;
Temp_INT[0]	:= RequestPickingListFromHMI[2].State; 						//Stato WO richiesto
Temp_UINT[0]:= RequestPickingListFromHMI[2].SlabNumber;			// Numero Lastre da depositare

// compilazione WO
// Tipologia: 0= Orrizzontale LEGNO,1= Orrizzontale Telaio , 2 = Bundle, 3 = A-FRAME
Temp_INT[0] := WorkareaState[1].Supporto.Tipologia;
Temp_INT[0] := WorkareaState[2].Supporto.Tipologia;
Temp_INT[0] := WorkareaState[3].Supporto.Tipologia;
Temp_INT[0] := WorkareaState[4].Supporto.Tipologia;
	//...	
Temp_INT[0] := WorkareaState[8].Supporto.Tipologia;

IF (FALSE) THEN
(*
// Per ogni Postazione
// Postazione 1	
//	HMI_WorkAreaDataPicking[1].Destinazione := 0;		//Prel/Depo
	HMI_WorkAreaDataPicking[1].Typology := 0;			//Cassa,Telaio,...
	HMI_WorkAreaDataPicking[1].NumElementiDaLavorare := 0; // Lastre da prelevare, se la Postazione è di deposito, SCOMPARE!
	HMI_NumeroLastreRimanentiOrdineAttuale[1] :=0;	
	HMI_WorkAreaDataPicking[1].NumElementiDaLavorare := 0; // dopo la Barra
	HMI_NumeroPezziPresentiPostazione[1] :=0;			//Campo sotto la cornice	
// Postazione 2	
	HMI_WorkAreaDataPicking[2].Destinazione := 0;		//Prel/Depo
	HMI_WorkAreaDataPicking[2].Typology := 0;			//Cassa,Telaio,...
	HMI_WorkAreaDataPicking[2].NumElementiDaLavorare := 0; // Lastre da prelevare, se la Postazione è di deposito, SCOMPARE!
	HMI_NumeroLastreRimanentiOrdineAttuale[2] :=0;	
	HMI_WorkAreaDataPicking[2].NumElementiDaLavorare := 0; // dopo la Barra
	HMI_NumeroPezziPresentiPostazione[2] :=0;			//Campo sotto la cornice	
// Postazione 3
	HMI_WorkAreaDataPicking[3].Destinazione := 0;		//Prel/Depo
	HMI_WorkAreaDataPicking[3].Typology := 0;			//Cassa,Telaio,...
	HMI_WorkAreaDataPicking[3].NumElementiDaLavorare := 0; // Lastre da prelevare, se la Postazione è di deposito, SCOMPARE!
	HMI_NumeroLastreRimanentiOrdineAttuale[3] :=0;
	HMI_WorkAreaDataPicking[3].NumElementiDaLavorare := 0; // dopo la Barra
	HMI_NumeroPezziPresentiPostazione[3] :=0;			//Campo sotto la cornice	


// Work Order Richiesto
	RequestPickingListFromHMI[2].State :=0;
	RequestPickingListFromHMI[2].SlabNumber :=0;
// Work Order attuale	
	ActualPickingListFromHMI[2].State  :=0;	
	HMI_NumeroLastreDepOrdineAttuale[2] :=0; 
	RequestPickingListFromHMI[2].SlabNumber :=0;
	
	ElementiDaDepositare[Temp_IdxLista]  := Temp_UINT[0]; //# Somma delle Lastre da Prelevare nelle WorkArea
	WorkAreaState[Temp_i].P := Temp_INT[0];				//# Pack Poinyer, contiene il NumElementiDaLavorare
	
	//Controllo sul numero elementi da prelevare che deve essere min o uguale agli elementi da depositare
	ActualPickingListFromHMI[Temp_IdxLista]	:= RequestPickingListFromHMI[Temp_IdxLista];
	ActualPickingListFromHMI[Temp_IdxLista].State 	:= e_StatoWorkOrder.DA_ESEGUIRE;
	
	Temp_INT[0] := Picking.RequestPickingListFromHMI[1].SupportPianoLegno.Code;
	Temp_INT[0]	:= RequestPickingListFromHMI[Temp_IdxLista].SupportPianoLegno.Code;
	Temp_REAL[0] := RequestPickingListFromHMI[Temp_IdxLista].SupportPianoLegno.XDim;
	Temp_REAL[0] := RequestPickingListFromHMI[Temp_IdxLista].SupportPianoLegno.YDim;
	Temp_REAL[0] := RequestPickingListFromHMI[Temp_IdxLista].SupportPianoLegno.ZDim;
	Temp_INT[3] := HMI_WorkAreaDataPicking[1].Typology;

	// Lista di produzione compilata
	//WorkAreaProductionList[MAXAREA].PElementList[MAXELEMENTLIST].WA_PRELIEVO :=0;
	//WorkAreaProductionList[MAXAREA].PElementList[MAXELEMENTLIST].WA_DEPOSITO :=0;
	
	//Work Area Production List 1
	WorkAreaProductionList[1].PElementList[1].WA_PRELIEVO :=0;
	WorkAreaProductionList[1].PElementList[2].WA_PRELIEVO :=0;
	WorkAreaProductionList[1].PElementList[3].WA_PRELIEVO :=0;
	
	WorkAreaProductionList[1].PElementList[1].WA_DEPOSITO :=0;
	WorkAreaProductionList[1].PElementList[2].WA_DEPOSITO :=0;
	WorkAreaProductionList[1].PElementList[3].WA_DEPOSITO :=0;
	//Work Area Production List 2	
	WorkAreaProductionList[2].PElementList[1].WA_PRELIEVO :=0;
	WorkAreaProductionList[2].PElementList[2].WA_PRELIEVO :=0;
	WorkAreaProductionList[2].PElementList[3].WA_PRELIEVO :=0;
	WorkAreaProductionList[2].PElementList[4].WA_PRELIEVO :=0;
	WorkAreaProductionList[2].PElementList[5].WA_PRELIEVO :=0;
		
	WorkAreaProductionList[2].PElementList[1].WA_DEPOSITO :=0;
	WorkAreaProductionList[2].PElementList[2].WA_DEPOSITO :=0;
	WorkAreaProductionList[2].PElementList[3].WA_DEPOSITO :=0;
	WorkAreaProductionList[2].PElementList[4].WA_DEPOSITO :=0;
	WorkAreaProductionList[2].PElementList[5].WA_DEPOSITO :=0;
//Work Area Production List 3 (WA dove viene fatto il prelievo con 5 lastre da spostare)
	WorkAreaProductionList[3].PElementList[1].WA_PRELIEVO :=0;
	WorkAreaProductionList[3].PElementList[2].WA_PRELIEVO :=0;
	WorkAreaProductionList[3].PElementList[3].WA_PRELIEVO :=0;
	WorkAreaProductionList[3].PElementList[4].WA_PRELIEVO :=0;
	WorkAreaProductionList[3].PElementList[5].WA_PRELIEVO :=0;
	WorkAreaProductionList[3].PElementList[6].WA_PRELIEVO :=0;
							 //(WA dove viene fatto il deposito con 5 lastre da spostare)
	WorkAreaProductionList[3].PElementList[1].WA_DEPOSITO :=0;
	WorkAreaProductionList[3].PElementList[2].WA_DEPOSITO :=0;
	WorkAreaProductionList[3].PElementList[3].WA_DEPOSITO :=0;
	WorkAreaProductionList[3].PElementList[4].WA_DEPOSITO :=0;
	WorkAreaProductionList[3].PElementList[5].WA_DEPOSITO :=0;
	WorkAreaProductionList[3].PElementList[6].WA_DEPOSITO :=0;
//Work Area Production List 4
	WorkAreaProductionList[4].PElementList[1].WA_PRELIEVO :=0;
	WorkAreaProductionList[4].PElementList[2].WA_PRELIEVO :=0;
	WorkAreaProductionList[4].PElementList[3].WA_PRELIEVO :=0;
	WorkAreaProductionList[4].PElementList[4].WA_PRELIEVO :=0;
	WorkAreaProductionList[4].PElementList[5].WA_PRELIEVO :=0;
		
	WorkAreaProductionList[4].PElementList[1].WA_DEPOSITO :=0;
	WorkAreaProductionList[4].PElementList[2].WA_DEPOSITO :=0;
	WorkAreaProductionList[4].PElementList[3].WA_DEPOSITO :=0;
	WorkAreaProductionList[4].PElementList[4].WA_DEPOSITO :=0;
	WorkAreaProductionList[4].PElementList[5].WA_DEPOSITO :=0;	
	
// TEST SE LISTA E' ATTIVATA
	ActualPickingListFromHMI[1].State :=0;//Ordine postazioni 1..8 in lavoro
	ActualPickingListFromHMI[2].State :=0;//Ordine postazioni 1..4 in lavoro
	ActualPickingListFromHMI[3].State :=0;//Ordine postazioni 5..8 in lavoro
		
	HMI_WorkAreaDataPicking_1_8 := 0;//Ordine postazioni 1..8 in lavoro
	HMI_WorkAreaDataPicking_1_4 := 0;//Ordine postazioni 1..4 in lavoro
	HMI_WorkAreaDataPicking_5_8 := 0;//Ordine postazioni 5..8 in lavoro
*)	
END_IF
END_ACTION

END_PROGRAM

(* stored: Version 1.1.0.1, ProductVersion 3.1.4024.11
   POU TFMachinePalletizerMain: Id {221e7216-b954-4275-985d-be09336b2a7f}, SpecialFunc None
   Action _01_Init: Id {fa3d889e-765b-4ab4-a788-a005a143d5ea}
   Action _02_LeggiInput: Id {0744d895-81b3-432e-8d3d-f3d6ef154f79}
   Action _03_Modules: Id {a611c0f7-588c-4abe-b290-7ee028a356b7}
   Action _04_Comunicazione: Id {69410ae8-a506-4ad3-ab4e-b4b673581bd0}
   Action _05_ManualCmds: Id {605028ed-4808-4ad5-96e5-b72daae2ec78}
   Action _06_ScriviOutput: Id {395db207-29a8-45db-b071-eb769af8bdaa}
   Action _07_ScriviStatus: Id {6cd47633-e11d-4337-903f-067cef6313cd}
   Action _08_DataLogger_ACT: Id {e7428516-cc17-4a9a-8206-fa2638885dc6}
   Action _09_CalcolaFormatura: Id {c2cfc39e-ed3a-4d30-b6b5-c2cbe6990a0b}
   Action _10_PackModifier: Id {fe2414cb-edd2-4aa8-a335-29a17133418c}
   Action _11_CalcolaListaProduzione: Id {b5a90fc5-183c-446d-9172-e9ebb125fccb}
   Action _11_CalcolaListaProduzioneold: Id {71f8cc26-c970-492d-8e1e-8fd09f70d1e6}
   Action TEST_Variabili: Id {d1477142-a8d1-4d92-b199-364b2f7edc0e} *)
